gfCNCPoint5[20423] = {X 281.5052, Y 41.6984, Z -7.1667, A 0.000, B 0.000, C 0.000 }
gfCNCPoint5[20424] = {X 282.1444, Y 41.0612, Z -7.1667, A 0.000, B 0.000, C 0.000 }
gfCNCPoint5[20425] = {X 282.1444, Y 28.5919, Z -7.1667, A 0.000, B 0.000, C 0.000 }
gfCNCPoint5[20426] = {X 278.0644, Y 28.5919, Z -7.1667, A 0.000, B 0.000, C 0.000 }
gfCNCPoint5[20427] = {X 278.0644, Y 28.5919, Z -4.1667, A 0.000, B 0.000, C 0.000 }
gfCNCPoint5[20428] = {X 278.0644, Y 28.5919, Z 11.0000, A 0.000, B 0.000, C 0.000 }
gfCNCPoint5[20429] = {X 353.3540, Y 107.0415, Z 11.0000, A 0.000, B 0.000, C 0.000 }
gfCNCPoint5[20430] = {X 353.3540, Y 107.0415, Z -4.1667, A 0.000, B 0.000, C 0.000 }
gfCNCPoint5[20431] = {X 353.3540, Y 107.0415, Z -7.1667, A 0.000, B 0.000, C 0.000 }
gfCNCPoint5[20432] = {X 353.2425, Y 102.9631, Z -7.1667, A 0.000, B 0.000, C 0.000 }
gfCNCPoint5[20433] = {X 348.1839, Y 103.0329, Z -7.1667, A 0.000, B 0.000, C 0.000 }
gfCNCPoint5[20434] = {X 343.1251, Y 102.9662, Z -7.1667, A 0.000, B 0.000, C 0.000 }
gfCNCPoint5[20435] = {X 338.0701, Y 102.7628, Z -7.1667, A 0.000, B 0.000, C 0.000 }
gfCNCPoint5[20436] = {X 334.1158, Y 102.4859, Z -7.1667, A 0.000, B 0.000, C 0.000 }
gfCNCPoint5[20437] = {X 330.1765, Y 102.0440, Z -7.1667, A 0.000, B 0.000, C 0.000 }
gfCNCPoint5[20438] = {X 326.2592, Y 101.4380, Z -7.1667, A 0.000, B 0.000, C 0.000 }
gfCNCPoint5[20439] = {X 323.4097, Y 100.8332, Z -7.1667, A 0.000, B 0.000, C 0.000 }
gfCNCPoint5[20440] = {X 320.6125, Y 100.0203, Z -7.1667, A 0.000, B 0.000, C 0.000 }
gfCNCPoint5[20441] = {X 317.8826, Y 99.0038, Z -7.1667, A 0.000, B 0.000, C 0.000 }
gfCNCPoint5[20442] = {X 316.3697, Y 98.3059, Z -7.1667, A 0.000, B 0.000, C 0.000 }
gfCNCPoint5[20443] = {X 314.9204, Y 97.4840, Z -7.1667, A 0.000, B 0.000, C 0.000 }
gfCNCPoint5[20444] = {X 313.5448, Y 96.5439, Z -7.1667, A 0.000, B 0.000, C 0.000 }
gfCNCPoint5[20445] = {X 312.2527, Y 95.4921, Z -7.1667, A 0.000, B 0.000, C 0.000 }
gfCNCPoint5[20446] = {X 311.2489, Y 94.4933, Z -7.1667, A 0.000, B 0.000, C 0.000 }
gfCNCPoint5[20447] = {X 310.3705, Y 93.3827, Z -7.1667, A 0.000, B 0.000, C 0.000 }
gfCNCPoint5[20448] = {X 309.6299, Y 92.1758, Z -7.1667, A 0.000, B 0.000, C 0.000 }
gfCNCPoint5[20449] = {X 309.0375, Y 90.8896, Z -7.1667, A 0.000, B 0.000, C 0.000 }
gfCNCPoint5[20450] = {X 308.6017, Y 89.5424, Z -7.1667, A 0.000, B 0.000, C 0.000 }
gfCNCPoint5[20451] = {X 308.2582, Y 87.9192, Z -7.1667, A 0.000, B 0.000, C 0.000 }
gfCNCPoint5[20452] = {X 308.0553, Y 86.2726, Z -7.1667, A 0.000, B 0.000, C 0.000 }
gfCNCPoint5[20453] = {X 307.9944, Y 84.6146, Z -7.1667, A 0.000, B 0.000, C 0.000 }
gfCNCPoint5[20454] = {X 307.9956, Y 63.2121, Z -7.1667, A 0.000, B 0.000, C 0.000 }
gfCNCPoint5[20455] = {X 307.1443, Y 63.0028, Z -7.1667, A 0.000, B 0.000, C 0.000 }
gfCNCPoint5[20456] = {X 306.3527, Y 62.6258, Z -7.1667, A 0.000, B 0.000, C 0.000 }
gfCNCPoint5[20457] = {X 305.6536, Y 62.0968, Z -7.1667, A 0.000, B 0.000, C 0.000 }
gfCNCPoint5[20458] = {X 305.0756, Y 61.4376, Z -7.1667, A 0.000, B 0.000, C 0.000 }
gfCNCPoint5[20459] = {X 304.6427, Y 60.6752, Z -7.1667, A 0.000, B 0.000, C 0.000 }
gfCNCPoint5[20460] = {X 304.3725, Y 59.8412, Z -7.1667, A 0.000, B 0.000, C 0.000 }
gfCNCPoint5[20461] = {X 304.2764, Y 58.9697, Z -7.1667, A 0.000, B 0.000, C 0.000 }
gfCNCPoint5[20462] = {X 304.2762, Y 58.0000, Z -7.1667, A 0.000, B 0.000, C 0.000 }
gfCNCPoint5[20463] = {X 304.3845, Y 57.0387, Z -7.1667, A 0.000, B 0.000, C 0.000 }
gfCNCPoint5[20464] = {X 304.7040, Y 56.1256, Z -7.1667, A 0.000, B 0.000, C 0.000 }
gfCNCPoint5[20465] = {X 305.2187, Y 55.3065, Z -7.1667, A 0.000, B 0.000, C 0.000 }
gfCNCPoint5[20466] = {X 305.9027, Y 54.6225, Z -7.1667, A 0.000, B 0.000, C 0.000 }
gfCNCPoint5[20467] = {X 306.7218, Y 54.1078, Z -7.1667, A 0.000, B 0.000, C 0.000 }
gfCNCPoint5[20468] = {X 307.6349, Y 53.7883, Z -7.1667, A 0.000, B 0.000, C 0.000 }
gfCNCPoint5[20469] = {X 308.5962, Y 53.6800, Z -7.1667, A 0.000, B 0.000, C 0.000 }
gfCNCPoint5[20470] = {X 324.3107, Y 53.6800, Z -7.1667, A 0.000, B 0.000, C 0.000 }
gfCNCPoint5[20471] = {X 325.2720, Y 53.7883, Z -7.1667, A 0.000, B 0.000, C 0.000 }
gfCNCPoint5[20472] = {X 326.1851, Y 54.1078, Z -7.1667, A 0.000, B 0.000, C 0.000 }
gfCNCPoint5[20473] = {X 327.0042, Y 54.6225, Z -7.1667, A 0.000, B 0.000, C 0.000 }
gfCNCPoint5[20474] = {X 327.6882, Y 55.3065, Z -7.1667, A 0.000, B 0.000, C 0.000 }
gfCNCPoint5[20475] = {X 328.2029, Y 56.1256, Z -7.1667, A 0.000, B 0.000, C 0.000 }
gfCNCPoint5[20476] = {X 328.5224, Y 57.0387, Z -7.1667, A 0.000, B 0.000, C 0.000 }
gfCNCPoint5[20477] = {X 328.6307, Y 58.0000, Z -7.1667, A 0.000, B 0.000, C 0.000 }
gfCNCPoint5[20478] = {X 328.6307, Y 58.9358, Z -7.1667, A 0.000, B 0.000, C 0.000 }
gfCNCPoint5[20479] = {X 328.5369, Y 59.8122, Z -7.1667, A 0.000, B 0.000, C 0.000 }
gfCNCPoint5[20480] = {X 328.2687, Y 60.6517, Z -7.1667, A 0.000, B 0.000, C 0.000 }
gfCNCPoint5[20481] = {X 327.8370, Y 61.4202, Z -7.1667, A 0.000, B 0.000, C 0.000 }
gfCNCPoint5[20482] = {X 327.2595, Y 62.0860, Z -7.1667, A 0.000, B 0.000, C 0.000 }
gfCNCPoint5[20483] = {X 326.5599, Y 62.6220, Z -7.1667, A 0.000, B 0.000, C 0.000 }
gfCNCPoint5[20484] = {X 325.7666, Y 63.0063, Z -7.1667, A 0.000, B 0.000, C 0.000 }
gfCNCPoint5[20485] = {X 324.9123, Y 63.2230, Z -7.1667, A 0.000, B 0.000, C 0.000 }
gfCNCPoint5[20486] = {X 324.9142, Y 83.2295, Z -7.1667, A 0.000, B 0.000, C 0.000 }
gfCNCPoint5[20487] = {X 324.9278, Y 84.6145, Z -7.1667, A 0.000, B 0.000, C 0.000 }
gfCNCPoint5[20488] = {X 325.0045, Y 85.8430, Z -7.1667, A 0.000, B 0.000, C 0.000 }
gfCNCPoint5[20489] = {X 325.2231, Y 87.0543, Z -7.1667, A 0.000, B 0.000, C 0.000 }
gfCNCPoint5[20490] = {X 325.6723, Y 87.4784, Z -7.1667, A 0.000, B 0.000, C 0.000 }
gfCNCPoint5[20491] = {X 326.2083, Y 87.7855, Z -7.1667, A 0.000, B 0.000, C 0.000 }
gfCNCPoint5[20492] = {X 327.9881, Y 88.4971, Z -7.1667, A 0.000, B 0.000, C 0.000 }
gfCNCPoint5[20493] = {X 329.8404, Y 88.9900, Z -7.1667, A 0.000, B 0.000, C 0.000 }
gfCNCPoint5[20494] = {X 332.9245, Y 89.5434, Z -7.1667, A 0.000, B 0.000, C 0.000 }
gfCNCPoint5[20495] = {X 336.0365, Y 89.9077, Z -7.1667, A 0.000, B 0.000, C 0.000 }
gfCNCPoint5[20496] = {X 340.4063, Y 90.2019, Z -7.1667, A 0.000, B 0.000, C 0.000 }
gfCNCPoint5[20497] = {X 344.7832, Y 90.3557, Z -7.1667, A 0.000, B 0.000, C 0.000 }
gfCNCPoint5[20498] = {X 349.1628, Y 90.3690, Z -7.1667, A 0.000, B 0.000, C 0.000 }
gfCNCPoint5[20499] = {X 353.3143, Y 90.3007, Z -7.1667, A 0.000, B 0.000, C 0.000 }
gfCNCPoint5[20500] = {X 357.4606, Y 90.0817, Z -7.1667, A 0.000, B 0.000, C 0.000 }
gfCNCPoint5[20501] = {X 361.5962, Y 89.7124, Z -7.1667, A 0.000, B 0.000, C 0.000 }
gfCNCPoint5[20502] = {X 363.6775, Y 89.4253, Z -7.1667, A 0.000, B 0.000, C 0.000 }
gfCNCPoint5[20503] = {X 365.7396, Y 89.0233, Z -7.1667, A 0.000, B 0.000, C 0.000 }
gfCNCPoint5[20504] = {X 367.7763, Y 88.5076, Z -7.1667, A 0.000, B 0.000, C 0.000 }
gfCNCPoint5[20505] = {X 368.7088, Y 88.1946, Z -7.1667, A 0.000, B 0.000, C 0.000 }
gfCNCPoint5[20506] = {X 369.6001, Y 87.7787, Z -7.1667, A 0.000, B 0.000, C 0.000 }
gfCNCPoint5[20507] = {X 370.4388, Y 87.2650, Z -7.1667, A 0.000, B 0.000, C 0.000 }
gfCNCPoint5[20508] = {X 370.5874, Y 87.1102, Z -7.1667, A 0.000, B 0.000, C 0.000 }
gfCNCPoint5[20509] = {X 370.6640, Y 86.9098, Z -7.1667, A 0.000, B 0.000, C 0.000 }
gfCNCPoint5[20510] = {X 370.8553, Y 85.3746, Z -7.1667, A 0.000, B 0.000, C 0.000 }
gfCNCPoint5[20511] = {X 370.9191, Y 83.8288, Z -7.1667, A 0.000, B 0.000, C 0.000 }
gfCNCPoint5[20512] = {X 370.9200, Y 63.2123, Z -7.1667, A 0.000, B 0.000, C 0.000 }
gfCNCPoint5[20513] = {X 370.0684, Y 63.0031, Z -7.1667, A 0.000, B 0.000, C 0.000 }
gfCNCPoint5[20514] = {X 369.2766, Y 62.6263, Z -7.1667, A 0.000, B 0.000, C 0.000 }
gfCNCPoint5[20515] = {X 368.5772, Y 62.0973, Z -7.1667, A 0.000, B 0.000, C 0.000 }
gfCNCPoint5[20516] = {X 367.9990, Y 61.4381, Z -7.1667, A 0.000, B 0.000, C 0.000 }
gfCNCPoint5[20517] = {X 367.5659, Y 60.6756, Z -7.1667, A 0.000, B 0.000, C 0.000 }
gfCNCPoint5[20518] = {X 367.2956, Y 59.8414, Z -7.1667, A 0.000, B 0.000, C 0.000 }
gfCNCPoint5[20519] = {X 367.1994, Y 58.9697, Z -7.1667, A 0.000, B 0.000, C 0.000 }
gfCNCPoint5[20520] = {X 367.1993, Y 58.0000, Z -7.1667, A 0.000, B 0.000, C 0.000 }
gfCNCPoint5[20521] = {X 367.3076, Y 57.0387, Z -7.1667, A 0.000, B 0.000, C 0.000 }
gfCNCPoint5[20522] = {X 367.6271, Y 56.1256, Z -7.1667, A 0.000, B 0.000, C 0.000 }
gfCNCPoint5[20523] = {X 368.1418, Y 55.3065, Z -7.1667, A 0.000, B 0.000, C 0.000 }
gfCNCPoint5[20524] = {X 368.8258, Y 54.6225, Z -7.1667, A 0.000, B 0.000, C 0.000 }
gfCNCPoint5[20525] = {X 369.6449, Y 54.1078, Z -7.1667, A 0.000, B 0.000, C 0.000 }
gfCNCPoint5[20526] = {X 370.5580, Y 53.7883, Z -7.1667, A 0.000, B 0.000, C 0.000 }
gfCNCPoint5[20527] = {X 371.5193, Y 53.6800, Z -7.1667, A 0.000, B 0.000, C 0.000 }
gfCNCPoint5[20528] = {X 388.0597, Y 53.6800, Z -7.1667, A 0.000, B 0.000, C 0.000 }
gfCNCPoint5[20529] = {X 389.0210, Y 53.7883, Z -7.1667, A 0.000, B 0.000, C 0.000 }
gfCNCPoint5[20530] = {X 389.9341, Y 54.1078, Z -7.1667, A 0.000, B 0.000, C 0.000 }
gfCNCPoint5[20531] = {X 390.7532, Y 54.6225, Z -7.1667, A 0.000, B 0.000, C 0.000 }
gfCNCPoint5[20532] = {X 391.4372, Y 55.3065, Z -7.1667, A 0.000, B 0.000, C 0.000 }
gfCNCPoint5[20533] = {X 391.9519, Y 56.1256, Z -7.1667, A 0.000, B 0.000, C 0.000 }
gfCNCPoint5[20534] = {X 392.2714, Y 57.0387, Z -7.1667, A 0.000, B 0.000, C 0.000 }
gfCNCPoint5[20535] = {X 392.3797, Y 58.0000, Z -7.1667, A 0.000, B 0.000, C 0.000 }
gfCNCPoint5[20536] = {X 392.3797, Y 58.9342, Z -7.1667, A 0.000, B 0.000, C 0.000 }
gfCNCPoint5[20537] = {X 392.2681, Y 59.9098, Z -7.1667, A 0.000, B 0.000, C 0.000 }
gfCNCPoint5[20538] = {X 391.9390, Y 60.8349, Z -7.1667, A 0.000, B 0.000, C 0.000 }
gfCNCPoint5[20539] = {X 391.4969, Y 61.5528, Z -7.1667, A 0.000, B 0.000, C 0.000 }
gfCNCPoint5[20540] = {X 390.9244, Y 62.1718, Z -7.1667, A 0.000, B 0.000, C 0.000 }
gfCNCPoint5[20541] = {X 390.2431, Y 62.6686, Z -7.1667, A 0.000, B 0.000, C 0.000 }
gfCNCPoint5[20542] = {X 389.4787, Y 63.0243, Z -7.1667, A 0.000, B 0.000, C 0.000 }
gfCNCPoint5[20543] = {X 388.6600, Y 63.2257, Z -7.1667, A 0.000, B 0.000, C 0.000 }
gfCNCPoint5[20544] = {X 388.6579, Y 84.6147, Z -7.1667, A 0.000, B 0.000, C 0.000 }
gfCNCPoint5[20545] = {X 388.5980, Y 86.2730, Z -7.1667, A 0.000, B 0.000, C 0.000 }
gfCNCPoint5[20546] = {X 388.3937, Y 87.9198, Z -7.1667, A 0.000, B 0.000, C 0.000 }
gfCNCPoint5[20547] = {X 388.0465, Y 89.5425, Z -7.1667, A 0.000, B 0.000, C 0.000 }
gfCNCPoint5[20548] = {X 387.5140, Y 91.1297, Z -7.1667, A 0.000, B 0.000, C 0.000 }
gfCNCPoint5[20549] = {X 386.7643, Y 92.6265, Z -7.1667, A 0.000, B 0.000, C 0.000 }
gfCNCPoint5[20550] = {X 385.8124, Y 94.0036, Z -7.1667, A 0.000, B 0.000, C 0.000 }
gfCNCPoint5[20551] = {X 384.6769, Y 95.2337, Z -7.1667, A 0.000, B 0.000, C 0.000 }
gfCNCPoint5[20552] = {X 383.1622, Y 96.5103, Z -7.1667, A 0.000, B 0.000, C 0.000 }
gfCNCPoint5[20553] = {X 381.5205, Y 97.6188, Z -7.1667, A 0.000, B 0.000, C 0.000 }
gfCNCPoint5[20554] = {X 379.7703, Y 98.5466, Z -7.1667, A 0.000, B 0.000, C 0.000 }
gfCNCPoint5[20555] = {X 377.4988, Y 99.5016, Z -7.1667, A 0.000, B 0.000, C 0.000 }
gfCNCPoint5[20556] = {X 375.1648, Y 100.2918, Z -7.1667, A 0.000, B 0.000, C 0.000 }
gfCNCPoint5[20557] = {X 372.7804, Y 100.9132, Z -7.1667, A 0.000, B 0.000, C 0.000 }
gfCNCPoint5[20558] = {X 368.8695, Y 101.6665, Z -7.1667, A 0.000, B 0.000, C 0.000 }
gfCNCPoint5[20559] = {X 364.9264, Y 102.2268, Z -7.1667, A 0.000, B 0.000, C 0.000 }
gfCNCPoint5[20560] = {X 360.9605, Y 102.5928, Z -7.1667, A 0.000, B 0.000, C 0.000 }
gfCNCPoint5[20561] = {X 357.1034, Y 102.8177, Z -7.1667, A 0.000, B 0.000, C 0.000 }
gfCNCPoint5[20562] = {X 353.2425, Y 102.9631, Z -7.1667, A 0.000, B 0.000, C 0.000 }
gfCNCPoint5[20563] = {X 353.3518, Y 106.9616, Z -7.1667, A 0.000, B 0.000, C 0.000 }
gfCNCPoint5[20564] = {X 353.2403, Y 102.8831, Z -7.1667, A 0.000, B 0.000, C 0.000 }
gfCNCPoint5[20565] = {X 348.1838, Y 102.9529, Z -7.1667, A 0.000, B 0.000, C 0.000 }
gfCNCPoint5[20566] = {X 343.1272, Y 102.8862, Z -7.1667, A 0.000, B 0.000, C 0.000 }
gfCNCPoint5[20567] = {X 338.0742, Y 102.6829, Z -7.1667, A 0.000, B 0.000, C 0.000 }
gfCNCPoint5[20568] = {X 334.1232, Y 102.4062, Z -7.1667, A 0.000, B 0.000, C 0.000 }
gfCNCPoint5[20569] = {X 330.1871, Y 101.9647, Z -7.1667, A 0.000, B 0.000, C 0.000 }
gfCNCPoint5[20570] = {X 326.2730, Y 101.3592, Z -7.1667, A 0.000, B 0.000, C 0.000 }
gfCNCPoint5[20571] = {X 323.4292, Y 100.7556, Z -7.1667, A 0.000, B 0.000, C 0.000 }
gfCNCPoint5[20572] = {X 320.6375, Y 99.9443, Z -7.1667, A 0.000, B 0.000, C 0.000 }
gfCNCPoint5[20573] = {X 317.9131, Y 98.9298, Z -7.1667, A 0.000, B 0.000, C 0.000 }
gfCNCPoint5[20574] = {X 316.4062, Y 98.2347, Z -7.1667, A 0.000, B 0.000, C 0.000 }
gfCNCPoint5[20575] = {X 314.9627, Y 97.4161, Z -7.1667, A 0.000, B 0.000, C 0.000 }
gfCNCPoint5[20576] = {X 313.5926, Y 96.4797, Z -7.1667, A 0.000, B 0.000, C 0.000 }
gfCNCPoint5[20577] = {X 312.3056, Y 95.4321, Z -7.1667, A 0.000, B 0.000, C 0.000 }
gfCNCPoint5[20578] = {X 311.3086, Y 94.4401, Z -7.1667, A 0.000, B 0.000, C 0.000 }
gfCNCPoint5[20579] = {X 310.4361, Y 93.3368, Z -7.1667, A 0.000, B 0.000, C 0.000 }
gfCNCPoint5[20580] = {X 309.7005, Y 92.1380, Z -7.1667, A 0.000, B 0.000, C 0.000 }
gfCNCPoint5[20581] = {X 309.1121, Y 90.8605, Z -7.1667, A 0.000, B 0.000, C 0.000 }
gfCNCPoint5[20582] = {X 308.6791, Y 89.5223, Z -7.1667, A 0.000, B 0.000, C 0.000 }
gfCNCPoint5[20583] = {X 308.3371, Y 87.9059, Z -7.1667, A 0.000, B 0.000, C 0.000 }
gfCNCPoint5[20584] = {X 308.1350, Y 86.2661, Z -7.1667, A 0.000, B 0.000, C 0.000 }
gfCNCPoint5[20585] = {X 308.0744, Y 84.6150, Z -7.1667, A 0.000, B 0.000, C 0.000 }
gfCNCPoint5[20586] = {X 308.0756, Y 63.1420, Z -7.1667, A 0.000, B 0.000, C 0.000 }
gfCNCPoint5[20587] = {X 307.2274, Y 62.9470, Z -7.1667, A 0.000, B 0.000, C 0.000 }
gfCNCPoint5[20588] = {X 306.4368, Y 62.5830, Z -7.1667, A 0.000, B 0.000, C 0.000 }
gfCNCPoint5[20589] = {X 305.7373, Y 62.0652, Z -7.1667, A 0.000, B 0.000, C 0.000 }
gfCNCPoint5[20590] = {X 305.1581, Y 61.4154, Z -7.1667, A 0.000, B 0.000, C 0.000 }
gfCNCPoint5[20591] = {X 304.7239, Y 60.6611, Z -7.1667, A 0.000, B 0.000, C 0.000 }
gfCNCPoint5[20592] = {X 304.4528, Y 59.8341, Z -7.1667, A 0.000, B 0.000, C 0.000 }
gfCNCPoint5[20593] = {X 304.3564, Y 58.9691, Z -7.1667, A 0.000, B 0.000, C 0.000 }
gfCNCPoint5[20594] = {X 304.3562, Y 58.0000, Z -7.1667, A 0.000, B 0.000, C 0.000 }
gfCNCPoint5[20595] = {X 304.4625, Y 57.0565, Z -7.1667, A 0.000, B 0.000, C 0.000 }
gfCNCPoint5[20596] = {X 304.7761, Y 56.1603, Z -7.1667, A 0.000, B 0.000, C 0.000 }
gfCNCPoint5[20597] = {X 305.2813, Y 55.3564, Z -7.1667, A 0.000, B 0.000, C 0.000 }
gfCNCPoint5[20598] = {X 305.9526, Y 54.6850, Z -7.1667, A 0.000, B 0.000, C 0.000 }
gfCNCPoint5[20599] = {X 306.7566, Y 54.1799, Z -7.1667, A 0.000, B 0.000, C 0.000 }
gfCNCPoint5[20600] = {X 307.6527, Y 53.8663, Z -7.1667, A 0.000, B 0.000, C 0.000 }
gfCNCPoint5[20601] = {X 308.5962, Y 53.7600, Z -7.1667, A 0.000, B 0.000, C 0.000 }
gfCNCPoint5[20602] = {X 324.3107, Y 53.7600, Z -7.1667, A 0.000, B 0.000, C 0.000 }
gfCNCPoint5[20603] = {X 325.2542, Y 53.8663, Z -7.1667, A 0.000, B 0.000, C 0.000 }
gfCNCPoint5[20604] = {X 326.1504, Y 54.1799, Z -7.1667, A 0.000, B 0.000, C 0.000 }
gfCNCPoint5[20605] = {X 326.9543, Y 54.6850, Z -7.1667, A 0.000, B 0.000, C 0.000 }
gfCNCPoint5[20606] = {X 327.6257, Y 55.3564, Z -7.1667, A 0.000, B 0.000, C 0.000 }
gfCNCPoint5[20607] = {X 328.1308, Y 56.1603, Z -7.1667, A 0.000, B 0.000, C 0.000 }
gfCNCPoint5[20608] = {X 328.4444, Y 57.0565, Z -7.1667, A 0.000, B 0.000, C 0.000 }
gfCNCPoint5[20609] = {X 328.5507, Y 58.0000, Z -7.1667, A 0.000, B 0.000, C 0.000 }
gfCNCPoint5[20610] = {X 328.5507, Y 58.9354, Z -7.1667, A 0.000, B 0.000, C 0.000 }
gfCNCPoint5[20611] = {X 328.4566, Y 59.8053, Z -7.1667, A 0.000, B 0.000, C 0.000 }
gfCNCPoint5[20612] = {X 328.1875, Y 60.6379, Z -7.1667, A 0.000, B 0.000, C 0.000 }
gfCNCPoint5[20613] = {X 327.7545, Y 61.3982, Z -7.1667, A 0.000, B 0.000, C 0.000 }
gfCNCPoint5[20614] = {X 327.1759, Y 62.0546, Z -7.1667, A 0.000, B 0.000, C 0.000 }
gfCNCPoint5[20615] = {X 326.4758, Y 62.5795, Z -7.1667, A 0.000, B 0.000, C 0.000 }
gfCNCPoint5[20616] = {X 325.6836, Y 62.9510, Z -7.1667, A 0.000, B 0.000, C 0.000 }
gfCNCPoint5[20617] = {X 324.8323, Y 63.1534, Z -7.1667, A 0.000, B 0.000, C 0.000 }
gfCNCPoint5[20618] = {X 324.8342, Y 83.2300, Z -7.1667, A 0.000, B 0.000, C 0.000 }
gfCNCPoint5[20619] = {X 324.8478, Y 84.6149, Z -7.1667, A 0.000, B 0.000, C 0.000 }
gfCNCPoint5[20620] = {X 324.9262, Y 85.8619, Z -7.1667, A 0.000, B 0.000, C 0.000 }
gfCNCPoint5[20621] = {X 325.1497, Y 87.0911, Z -7.1667, A 0.000, B 0.000, C 0.000 }
gfCNCPoint5[20622] = {X 325.6165, Y 87.5366, Z -7.1667, A 0.000, B 0.000, C 0.000 }
gfCNCPoint5[20623] = {X 326.1756, Y 87.8585, Z -7.1667, A 0.000, B 0.000, C 0.000 }
gfCNCPoint5[20624] = {X 327.9636, Y 88.5733, Z -7.1667, A 0.000, B 0.000, C 0.000 }
gfCNCPoint5[20625] = {X 329.8245, Y 89.0685, Z -7.1667, A 0.000, B 0.000, C 0.000 }
gfCNCPoint5[20626] = {X 332.9131, Y 89.6226, Z -7.1667, A 0.000, B 0.000, C 0.000 }
gfCNCPoint5[20627] = {X 336.0297, Y 89.9874, Z -7.1667, A 0.000, B 0.000, C 0.000 }
gfCNCPoint5[20628] = {X 340.4020, Y 90.2818, Z -7.1667, A 0.000, B 0.000, C 0.000 }
gfCNCPoint5[20629] = {X 344.7816, Y 90.4357, Z -7.1667, A 0.000, B 0.000, C 0.000 }
gfCNCPoint5[20630] = {X 349.1638, Y 90.4490, Z -7.1667, A 0.000, B 0.000, C 0.000 }
gfCNCPoint5[20631] = {X 353.3179, Y 90.3806, Z -7.1667, A 0.000, B 0.000, C 0.000 }
gfCNCPoint5[20632] = {X 357.4668, Y 90.1615, Z -7.1667, A 0.000, B 0.000, C 0.000 }
gfCNCPoint5[20633] = {X 361.6050, Y 89.7919, Z -7.1667, A 0.000, B 0.000, C 0.000 }
gfCNCPoint5[20634] = {X 363.6906, Y 89.5042, Z -7.1667, A 0.000, B 0.000, C 0.000 }
gfCNCPoint5[20635] = {X 365.7571, Y 89.1014, Z -7.1667, A 0.000, B 0.000, C 0.000 }
gfCNCPoint5[20636] = {X 367.7981, Y 88.5846, Z -7.1667, A 0.000, B 0.000, C 0.000 }
gfCNCPoint5[20637] = {X 368.7389, Y 88.2688, Z -7.1667, A 0.000, B 0.000, C 0.000 }
gfCNCPoint5[20638] = {X 369.6381, Y 87.8490, Z -7.1667, A 0.000, B 0.000, C 0.000 }
gfCNCPoint5[20639] = {X 370.4844, Y 87.3307, Z -7.1667, A 0.000, B 0.000, C 0.000 }
gfCNCPoint5[20640] = {X 370.6550, Y 87.1530, Z -7.1667, A 0.000, B 0.000, C 0.000 }
gfCNCPoint5[20641] = {X 370.7429, Y 86.9229, Z -7.1667, A 0.000, B 0.000, C 0.000 }
gfCNCPoint5[20642] = {X 370.9350, Y 85.3812, Z -7.1667, A 0.000, B 0.000, C 0.000 }
gfCNCPoint5[20643] = {X 370.9991, Y 83.8288, Z -7.1667, A 0.000, B 0.000, C 0.000 }
gfCNCPoint5[20644] = {X 371.0000, Y 63.1421, Z -7.1667, A 0.000, B 0.000, C 0.000 }
gfCNCPoint5[20645] = {X 370.1515, Y 62.9474, Z -7.1667, A 0.000, B 0.000, C 0.000 }
gfCNCPoint5[20646] = {X 369.3607, Y 62.5835, Z -7.1667, A 0.000, B 0.000, C 0.000 }
gfCNCPoint5[20647] = {X 368.6609, Y 62.0657, Z -7.1667, A 0.000, B 0.000, C 0.000 }
gfCNCPoint5[20648] = {X 368.0815, Y 61.4159, Z -7.1667, A 0.000, B 0.000, C 0.000 }
gfCNCPoint5[20649] = {X 367.6471, Y 60.6615, Z -7.1667, A 0.000, B 0.000, C 0.000 }
gfCNCPoint5[20650] = {X 367.3759, Y 59.8343, Z -7.1667, A 0.000, B 0.000, C 0.000 }
gfCNCPoint5[20651] = {X 367.2794, Y 58.9691, Z -7.1667, A 0.000, B 0.000, C 0.000 }
gfCNCPoint5[20652] = {X 367.2793, Y 58.0000, Z -7.1667, A 0.000, B 0.000, C 0.000 }
gfCNCPoint5[20653] = {X 367.3856, Y 57.0565, Z -7.1667, A 0.000, B 0.000, C 0.000 }
gfCNCPoint5[20654] = {X 367.6992, Y 56.1603, Z -7.1667, A 0.000, B 0.000, C 0.000 }
gfCNCPoint5[20655] = {X 368.2043, Y 55.3564, Z -7.1667, A 0.000, B 0.000, C 0.000 }
gfCNCPoint5[20656] = {X 368.8757, Y 54.6850, Z -7.1667, A 0.000, B 0.000, C 0.000 }
gfCNCPoint5[20657] = {X 369.6796, Y 54.1799, Z -7.1667, A 0.000, B 0.000, C 0.000 }
gfCNCPoint5[20658] = {X 370.5758, Y 53.8663, Z -7.1667, A 0.000, B 0.000, C 0.000 }
gfCNCPoint5[20659] = {X 371.5193, Y 53.7600, Z -7.1667, A 0.000, B 0.000, C 0.000 }
gfCNCPoint5[20660] = {X 388.0597, Y 53.7600, Z -7.1667, A 0.000, B 0.000, C 0.000 }
gfCNCPoint5[20661] = {X 389.0032, Y 53.8663, Z -7.1667, A 0.000, B 0.000, C 0.000 }
gfCNCPoint5[20662] = {X 389.8993, Y 54.1799, Z -7.1667, A 0.000, B 0.000, C 0.000 }
gfCNCPoint5[20663] = {X 390.7033, Y 54.6850, Z -7.1667, A 0.000, B 0.000, C 0.000 }
gfCNCPoint5[20664] = {X 391.3746, Y 55.3564, Z -7.1667, A 0.000, B 0.000, C 0.000 }
gfCNCPoint5[20665] = {X 391.8798, Y 56.1603, Z -7.1667, A 0.000, B 0.000, C 0.000 }
gfCNCPoint5[20666] = {X 392.1934, Y 57.0565, Z -7.1667, A 0.000, B 0.000, C 0.000 }
gfCNCPoint5[20667] = {X 392.2997, Y 58.0000, Z -7.1667, A 0.000, B 0.000, C 0.000 }
gfCNCPoint5[20668] = {X 392.2997, Y 58.9342, Z -7.1667, A 0.000, B 0.000, C 0.000 }
gfCNCPoint5[20669] = {X 392.1901, Y 59.8917, Z -7.1667, A 0.000, B 0.000, C 0.000 }
gfCNCPoint5[20670] = {X 391.8672, Y 60.7997, Z -7.1667, A 0.000, B 0.000, C 0.000 }
gfCNCPoint5[20671] = {X 391.4248, Y 61.5154, Z -7.1667, A 0.000, B 0.000, C 0.000 }
gfCNCPoint5[20672] = {X 390.8506, Y 62.1304, Z -7.1667, A 0.000, B 0.000, C 0.000 }
gfCNCPoint5[20673] = {X 390.1667, Y 62.6205, Z -7.1667, A 0.000, B 0.000, C 0.000 }
gfCNCPoint5[20674] = {X 389.3999, Y 62.9669, Z -7.1667, A 0.000, B 0.000, C 0.000 }
gfCNCPoint5[20675] = {X 388.5800, Y 63.1559, Z -7.1667, A 0.000, B 0.000, C 0.000 }
gfCNCPoint5[20676] = {X 388.5779, Y 84.6150, Z -7.1667, A 0.000, B 0.000, C 0.000 }
gfCNCPoint5[20677] = {X 388.5183, Y 86.2665, Z -7.1667, A 0.000, B 0.000, C 0.000 }
gfCNCPoint5[20678] = {X 388.3148, Y 87.9064, Z -7.1667, A 0.000, B 0.000, C 0.000 }
gfCNCPoint5[20679] = {X 387.9691, Y 89.5224, Z -7.1667, A 0.000, B 0.000, C 0.000 }
gfCNCPoint5[20680] = {X 387.4401, Y 91.0989, Z -7.1667, A 0.000, B 0.000, C 0.000 }
gfCNCPoint5[20681] = {X 386.6955, Y 92.5857, Z -7.1667, A 0.000, B 0.000, C 0.000 }
gfCNCPoint5[20682] = {X 385.7500, Y 93.9536, Z -7.1667, A 0.000, B 0.000, C 0.000 }
gfCNCPoint5[20683] = {X 384.6221, Y 95.1754, Z -7.1667, A 0.000, B 0.000, C 0.000 }
gfCNCPoint5[20684] = {X 383.1139, Y 96.4465, Z -7.1667, A 0.000, B 0.000, C 0.000 }
gfCNCPoint5[20685] = {X 381.4793, Y 97.5502, Z -7.1667, A 0.000, B 0.000, C 0.000 }
gfCNCPoint5[20686] = {X 379.7366, Y 98.4740, Z -7.1667, A 0.000, B 0.000, C 0.000 }
gfCNCPoint5[20687] = {X 377.4704, Y 99.4268, Z -7.1667, A 0.000, B 0.000, C 0.000 }
gfCNCPoint5[20688] = {X 375.1419, Y 100.2151, Z -7.1667, A 0.000, B 0.000, C 0.000 }
gfCNCPoint5[20689] = {X 372.7630, Y 100.8351, Z -7.1667, A 0.000, B 0.000, C 0.000 }
gfCNCPoint5[20690] = {X 368.8561, Y 101.5876, Z -7.1667, A 0.000, B 0.000, C 0.000 }
gfCNCPoint5[20691] = {X 364.9169, Y 102.1473, Z -7.1667, A 0.000, B 0.000, C 0.000 }
gfCNCPoint5[20692] = {X 360.9550, Y 102.5130, Z -7.1667, A 0.000, B 0.000, C 0.000 }
gfCNCPoint5[20693] = {X 357.0996, Y 102.7378, Z -7.1667, A 0.000, B 0.000, C 0.000 }
gfCNCPoint5[20694] = {X 353.2403, Y 102.8831, Z -7.1667, A 0.000, B 0.000, C 0.000 }
gfCNCPoint5[20695] = {X 353.3496, Y 106.8816, Z -7.1667, A 0.000, B 0.000, C 0.000 }
gfCNCPoint5[20696] = {X 353.2382, Y 102.8031, Z -7.1667, A 0.000, B 0.000, C 0.000 }
gfCNCPoint5[20697] = {X 348.1837, Y 102.8729, Z -7.1667, A 0.000, B 0.000, C 0.000 }
gfCNCPoint5[20698] = {X 343.1292, Y 102.8062, Z -7.1667, A 0.000, B 0.000, C 0.000 }
gfCNCPoint5[20699] = {X 338.0783, Y 102.6030, Z -7.1667, A 0.000, B 0.000, C 0.000 }
gfCNCPoint5[20700] = {X 334.1305, Y 102.3266, Z -7.1667, A 0.000, B 0.000, C 0.000 }
gfCNCPoint5[20701] = {X 330.1977, Y 101.8854, Z -7.1667, A 0.000, B 0.000, C 0.000 }
gfCNCPoint5[20702] = {X 326.2868, Y 101.2804, Z -7.1667, A 0.000, B 0.000, C 0.000 }
gfCNCPoint5[20703] = {X 323.4487, Y 100.6780, Z -7.1667, A 0.000, B 0.000, C 0.000 }
gfCNCPoint5[20704] = {X 320.6626, Y 99.8683, Z -7.1667, A 0.000, B 0.000, C 0.000 }
gfCNCPoint5[20705] = {X 317.9436, Y 98.8558, Z -7.1667, A 0.000, B 0.000, C 0.000 }
gfCNCPoint5[20706] = {X 316.4427, Y 98.1635, Z -7.1667, A 0.000, B 0.000, C 0.000 }
gfCNCPoint5[20707] = {X 315.0050, Y 97.3482, Z -7.1667, A 0.000, B 0.000, C 0.000 }
gfCNCPoint5[20708] = {X 313.6404, Y 96.4156, Z -7.1667, A 0.000, B 0.000, C 0.000 }
gfCNCPoint5[20709] = {X 312.3586, Y 95.3722, Z -7.1667, A 0.000, B 0.000, C 0.000 }
gfCNCPoint5[20710] = {X 311.3683, Y 94.3868, Z -7.1667, A 0.000, B 0.000, C 0.000 }
gfCNCPoint5[20711] = {X 310.5017, Y 93.2910, Z -7.1667, A 0.000, B 0.000, C 0.000 }
gfCNCPoint5[20712] = {X 309.7710, Y 92.1003, Z -7.1667, A 0.000, B 0.000, C 0.000 }
gfCNCPoint5[20713] = {X 309.1866, Y 90.8314, Z -7.1667, A 0.000, B 0.000, C 0.000 }
gfCNCPoint5[20714] = {X 308.7565, Y 89.5023, Z -7.1667, A 0.000, B 0.000, C 0.000 }
gfCNCPoint5[20715] = {X 308.4159, Y 87.8925, Z -7.1667, A 0.000, B 0.000, C 0.000 }
gfCNCPoint5[20716] = {X 308.2147, Y 86.2595, Z -7.1667, A 0.000, B 0.000, C 0.000 }
gfCNCPoint5[20717] = {X 308.1544, Y 84.6152, Z -7.1667, A 0.000, B 0.000, C 0.000 }
gfCNCPoint5[20718] = {X 308.1556, Y 63.0707, Z -7.1667, A 0.000, B 0.000, C 0.000 }
gfCNCPoint5[20719] = {X 307.3107, Y 62.8904, Z -7.1667, A 0.000, B 0.000, C 0.000 }
gfCNCPoint5[20720] = {X 306.5212, Y 62.5396, Z -7.1667, A 0.000, B 0.000, C 0.000 }
gfCNCPoint5[20721] = {X 305.8211, Y 62.0332, Z -7.1667, A 0.000, B 0.000, C 0.000 }
gfCNCPoint5[20722] = {X 305.2408, Y 61.3931, Z -7.1667, A 0.000, B 0.000, C 0.000 }
gfCNCPoint5[20723] = {X 304.8052, Y 60.6470, Z -7.1667, A 0.000, B 0.000, C 0.000 }
gfCNCPoint5[20724] = {X 304.5332, Y 59.8270, Z -7.1667, A 0.000, B 0.000, C 0.000 }
gfCNCPoint5[20725] = {X 304.4364, Y 58.9684, Z -7.1667, A 0.000, B 0.000, C 0.000 }
gfCNCPoint5[20726] = {X 304.4362, Y 58.0000, Z -7.1667, A 0.000, B 0.000, C 0.000 }
gfCNCPoint5[20727] = {X 304.5405, Y 57.0743, Z -7.1667, A 0.000, B 0.000, C 0.000 }
gfCNCPoint5[20728] = {X 304.8482, Y 56.1950, Z -7.1667, A 0.000, B 0.000, C 0.000 }
gfCNCPoint5[20729] = {X 305.3438, Y 55.4063, Z -7.1667, A 0.000, B 0.000, C 0.000 }
gfCNCPoint5[20730] = {X 306.0025, Y 54.7476, Z -7.1667, A 0.000, B 0.000, C 0.000 }
gfCNCPoint5[20731] = {X 306.7913, Y 54.2520, Z -7.1667, A 0.000, B 0.000, C 0.000 }
gfCNCPoint5[20732] = {X 307.6705, Y 53.9443, Z -7.1667, A 0.000, B 0.000, C 0.000 }
gfCNCPoint5[20733] = {X 308.5962, Y 53.8400, Z -7.1667, A 0.000, B 0.000, C 0.000 }
gfCNCPoint5[20734] = {X 324.3107, Y 53.8400, Z -7.1667, A 0.000, B 0.000, C 0.000 }
gfCNCPoint5[20735] = {X 325.2364, Y 53.9443, Z -7.1667, A 0.000, B 0.000, C 0.000 }
gfCNCPoint5[20736] = {X 326.1156, Y 54.2520, Z -7.1667, A 0.000, B 0.000, C 0.000 }
gfCNCPoint5[20737] = {X 326.9044, Y 54.7476, Z -7.1667, A 0.000, B 0.000, C 0.000 }
gfCNCPoint5[20738] = {X 327.5631, Y 55.4063, Z -7.1667, A 0.000, B 0.000, C 0.000 }
gfCNCPoint5[20739] = {X 328.0587, Y 56.1950, Z -7.1667, A 0.000, B 0.000, C 0.000 }
gfCNCPoint5[20740] = {X 328.3664, Y 57.0743, Z -7.1667, A 0.000, B 0.000, C 0.000 }
gfCNCPoint5[20741] = {X 328.4707, Y 58.0000, Z -7.1667, A 0.000, B 0.000, C 0.000 }
gfCNCPoint5[20742] = {X 328.4707, Y 58.9349, Z -7.1667, A 0.000, B 0.000, C 0.000 }
gfCNCPoint5[20743] = {X 328.3763, Y 59.7984, Z -7.1667, A 0.000, B 0.000, C 0.000 }
gfCNCPoint5[20744] = {X 328.1061, Y 60.6239, Z -7.1667, A 0.000, B 0.000, C 0.000 }
gfCNCPoint5[20745] = {X 327.6719, Y 61.3761, Z -7.1667, A 0.000, B 0.000, C 0.000 }
gfCNCPoint5[20746] = {X 327.0921, Y 62.0229, Z -7.1667, A 0.000, B 0.000, C 0.000 }
gfCNCPoint5[20747] = {X 326.3916, Y 62.5365, Z -7.1667, A 0.000, B 0.000, C 0.000 }
gfCNCPoint5[20748] = {X 325.6004, Y 62.8948, Z -7.1667, A 0.000, B 0.000, C 0.000 }
gfCNCPoint5[20749] = {X 324.7523, Y 63.0827, Z -7.1667, A 0.000, B 0.000, C 0.000 }
gfCNCPoint5[20750] = {X 324.7542, Y 83.2304, Z -7.1667, A 0.000, B 0.000, C 0.000 }
gfCNCPoint5[20751] = {X 324.7678, Y 84.6152, Z -7.1667, A 0.000, B 0.000, C 0.000 }
gfCNCPoint5[20752] = {X 324.8479, Y 85.8806, Z -7.1667, A 0.000, B 0.000, C 0.000 }
gfCNCPoint5[20753] = {X 325.0763, Y 87.1277, Z -7.1667, A 0.000, B 0.000, C 0.000 }
gfCNCPoint5[20754] = {X 325.5606, Y 87.5946, Z -7.1667, A 0.000, B 0.000, C 0.000 }
gfCNCPoint5[20755] = {X 326.1428, Y 87.9315, Z -7.1667, A 0.000, B 0.000, C 0.000 }
gfCNCPoint5[20756] = {X 327.9392, Y 88.6494, Z -7.1667, A 0.000, B 0.000, C 0.000 }
gfCNCPoint5[20757] = {X 329.8086, Y 89.1469, Z -7.1667, A 0.000, B 0.000, C 0.000 }
gfCNCPoint5[20758] = {X 332.9017, Y 89.7017, Z -7.1667, A 0.000, B 0.000, C 0.000 }
gfCNCPoint5[20759] = {X 336.0229, Y 90.0671, Z -7.1667, A 0.000, B 0.000, C 0.000 }
gfCNCPoint5[20760] = {X 340.3978, Y 90.3617, Z -7.1667, A 0.000, B 0.000, C 0.000 }
gfCNCPoint5[20761] = {X 344.7800, Y 90.5157, Z -7.1667, A 0.000, B 0.000, C 0.000 }
gfCNCPoint5[20762] = {X 349.1649, Y 90.5290, Z -7.1667, A 0.000, B 0.000, C 0.000 }
gfCNCPoint5[20763] = {X 353.3215, Y 90.4605, Z -7.1667, A 0.000, B 0.000, C 0.000 }
gfCNCPoint5[20764] = {X 357.4730, Y 90.2412, Z -7.1667, A 0.000, B 0.000, C 0.000 }
gfCNCPoint5[20765] = {X 361.6137, Y 89.8714, Z -7.1667, A 0.000, B 0.000, C 0.000 }
gfCNCPoint5[20766] = {X 363.7037, Y 89.5831, Z -7.1667, A 0.000, B 0.000, C 0.000 }
gfCNCPoint5[20767] = {X 365.7746, Y 89.1794, Z -7.1667, A 0.000, B 0.000, C 0.000 }
gfCNCPoint5[20768] = {X 367.8199, Y 88.6616, Z -7.1667, A 0.000, B 0.000, C 0.000 }
gfCNCPoint5[20769] = {X 368.7690, Y 88.3429, Z -7.1667, A 0.000, B 0.000, C 0.000 }
gfCNCPoint5[20770] = {X 369.6762, Y 87.9194, Z -7.1667, A 0.000, B 0.000, C 0.000 }
gfCNCPoint5[20771] = {X 370.5300, Y 87.3965, Z -7.1667, A 0.000, B 0.000, C 0.000 }
gfCNCPoint5[20772] = {X 370.7225, Y 87.1958, Z -7.1667, A 0.000, B 0.000, C 0.000 }
gfCNCPoint5[20773] = {X 370.8218, Y 86.9361, Z -7.1667, A 0.000, B 0.000, C 0.000 }
gfCNCPoint5[20774] = {X 371.0147, Y 85.3878, Z -7.1667, A 0.000, B 0.000, C 0.000 }
gfCNCPoint5[20775] = {X 371.0791, Y 83.8288, Z -7.1667, A 0.000, B 0.000, C 0.000 }
gfCNCPoint5[20776] = {X 371.0800, Y 63.0708, Z -7.1667, A 0.000, B 0.000, C 0.000 }
gfCNCPoint5[20777] = {X 370.9773, Y 63.0586, Z -7.1667, A 0.000, B 0.000, C 0.000 }
gfCNCPoint5[20778] = {X 370.8750, Y 63.0439, Z -7.1667, A 0.000, B 0.000, C 0.000 }
gfCNCPoint5[20779] = {X 369.9377, Y 62.7817, Z -7.1667, A 0.000, B 0.000, C 0.000 }
gfCNCPoint5[20780] = {X 369.0869, Y 62.3089, Z -7.1667, A 0.000, B 0.000, C 0.000 }
gfCNCPoint5[20781] = {X 368.3693, Y 61.6513, Z -7.1667, A 0.000, B 0.000, C 0.000 }
gfCNCPoint5[20782] = {X 367.8242, Y 60.8450, Z -7.1667, A 0.000, B 0.000, C 0.000 }
gfCNCPoint5[20783] = {X 367.4813, Y 59.9341, Z -7.1667, A 0.000, B 0.000, C 0.000 }
gfCNCPoint5[20784] = {X 367.3594, Y 58.9684, Z -7.1667, A 0.000, B 0.000, C 0.000 }
gfCNCPoint5[20785] = {X 367.3593, Y 58.0000, Z -7.1667, A 0.000, B 0.000, C 0.000 }
gfCNCPoint5[20786] = {X 367.4636, Y 57.0743, Z -7.1667, A 0.000, B 0.000, C 0.000 }
gfCNCPoint5[20787] = {X 367.7713, Y 56.1950, Z -7.1667, A 0.000, B 0.000, C 0.000 }
gfCNCPoint5[20788] = {X 368.2669, Y 55.4063, Z -7.1667, A 0.000, B 0.000, C 0.000 }
gfCNCPoint5[20789] = {X 368.9256, Y 54.7476, Z -7.1667, A 0.000, B 0.000, C 0.000 }
gfCNCPoint5[20790] = {X 369.7143, Y 54.2520, Z -7.1667, A 0.000, B 0.000, C 0.000 }
gfCNCPoint5[20791] = {X 370.5936, Y 53.9443, Z -7.1667, A 0.000, B 0.000, C 0.000 }
gfCNCPoint5[20792] = {X 371.5193, Y 53.8400, Z -7.1667, A 0.000, B 0.000, C 0.000 }
gfCNCPoint5[20793] = {X 388.0597, Y 53.8400, Z -7.1667, A 0.000, B 0.000, C 0.000 }
gfCNCPoint5[20794] = {X 388.9854, Y 53.9443, Z -7.1667, A 0.000, B 0.000, C 0.000 }
gfCNCPoint5[20795] = {X 389.8646, Y 54.2520, Z -7.1667, A 0.000, B 0.000, C 0.000 }
gfCNCPoint5[20796] = {X 390.6534, Y 54.7476, Z -7.1667, A 0.000, B 0.000, C 0.000 }
gfCNCPoint5[20797] = {X 391.3121, Y 55.4063, Z -7.1667, A 0.000, B 0.000, C 0.000 }
gfCNCPoint5[20798] = {X 391.8077, Y 56.1950, Z -7.1667, A 0.000, B 0.000, C 0.000 }
gfCNCPoint5[20799] = {X 392.1154, Y 57.0743, Z -7.1667, A 0.000, B 0.000, C 0.000 }
gfCNCPoint5[20800] = {X 392.2197, Y 58.0000, Z -7.1667, A 0.000, B 0.000, C 0.000 }
gfCNCPoint5[20801] = {X 392.2197, Y 58.9342, Z -7.1667, A 0.000, B 0.000, C 0.000 }
gfCNCPoint5[20802] = {X 392.1122, Y 59.8736, Z -7.1667, A 0.000, B 0.000, C 0.000 }
gfCNCPoint5[20803] = {X 391.7953, Y 60.7645, Z -7.1667, A 0.000, B 0.000, C 0.000 }
gfCNCPoint5[20804] = {X 391.2528, Y 61.6015, Z -7.1667, A 0.000, B 0.000, C 0.000 }
gfCNCPoint5[20805] = {X 390.5276, Y 62.2862, Z -7.1667, A 0.000, B 0.000, C 0.000 }
gfCNCPoint5[20806] = {X 389.6609, Y 62.7799, Z -7.1667, A 0.000, B 0.000, C 0.000 }
gfCNCPoint5[20807] = {X 388.7019, Y 63.0543, Z -7.1667, A 0.000, B 0.000, C 0.000 }
gfCNCPoint5[20808] = {X 388.6017, Y 63.0692, Z -7.1667, A 0.000, B 0.000, C 0.000 }
gfCNCPoint5[20809] = {X 388.5011, Y 63.0816, Z -7.1667, A 0.000, B 0.000, C 0.000 }
gfCNCPoint5[20810] = {X 388.4979, Y 84.6154, Z -7.1667, A 0.000, B 0.000, C 0.000 }
gfCNCPoint5[20811] = {X 388.4386, Y 86.2600, Z -7.1667, A 0.000, B 0.000, C 0.000 }
gfCNCPoint5[20812] = {X 388.2359, Y 87.8931, Z -7.1667, A 0.000, B 0.000, C 0.000 }
gfCNCPoint5[20813] = {X 387.8916, Y 89.5023, Z -7.1667, A 0.000, B 0.000, C 0.000 }
gfCNCPoint5[20814] = {X 387.3663, Y 91.0682, Z -7.1667, A 0.000, B 0.000, C 0.000 }
gfCNCPoint5[20815] = {X 386.6267, Y 92.5450, Z -7.1667, A 0.000, B 0.000, C 0.000 }
gfCNCPoint5[20816] = {X 385.6875, Y 93.9036, Z -7.1667, A 0.000, B 0.000, C 0.000 }
gfCNCPoint5[20817] = {X 384.5673, Y 95.1172, Z -7.1667, A 0.000, B 0.000, C 0.000 }
gfCNCPoint5[20818] = {X 383.0656, Y 96.3827, Z -7.1667, A 0.000, B 0.000, C 0.000 }
gfCNCPoint5[20819] = {X 381.4381, Y 97.4816, Z -7.1667, A 0.000, B 0.000, C 0.000 }
gfCNCPoint5[20820] = {X 379.7030, Y 98.4014, Z -7.1667, A 0.000, B 0.000, C 0.000 }
gfCNCPoint5[20821] = {X 377.4420, Y 99.3520, Z -7.1667, A 0.000, B 0.000, C 0.000 }
gfCNCPoint5[20822] = {X 375.1189, Y 100.1385, Z -7.1667, A 0.000, B 0.000, C 0.000 }
gfCNCPoint5[20823] = {X 372.7456, Y 100.7571, Z -7.1667, A 0.000, B 0.000, C 0.000 }
gfCNCPoint5[20824] = {X 368.8426, Y 101.5088, Z -7.1667, A 0.000, B 0.000, C 0.000 }
gfCNCPoint5[20825] = {X 364.9074, Y 102.0679, Z -7.1667, A 0.000, B 0.000, C 0.000 }
gfCNCPoint5[20826] = {X 360.9496, Y 102.4332, Z -7.1667, A 0.000, B 0.000, C 0.000 }
gfCNCPoint5[20827] = {X 357.0958, Y 102.6579, Z -7.1667, A 0.000, B 0.000, C 0.000 }
gfCNCPoint5[20828] = {X 353.2382, Y 102.8031, Z -7.1667, A 0.000, B 0.000, C 0.000 }
gfCNCPoint5[20829] = {X 353.3474, Y 106.8016, Z -7.1667, A 0.000, B 0.000, C 0.000 }
gfCNCPoint5[20830] = {X 353.2360, Y 102.7232, Z -7.1667, A 0.000, B 0.000, C 0.000 }
gfCNCPoint5[20831] = {X 348.1836, Y 102.7929, Z -7.1667, A 0.000, B 0.000, C 0.000 }
gfCNCPoint5[20832] = {X 343.1312, Y 102.7262, Z -7.1667, A 0.000, B 0.000, C 0.000 }
gfCNCPoint5[20833] = {X 338.0825, Y 102.5231, Z -7.1667, A 0.000, B 0.000, C 0.000 }
gfCNCPoint5[20834] = {X 334.1379, Y 102.2469, Z -7.1667, A 0.000, B 0.000, C 0.000 }
gfCNCPoint5[20835] = {X 330.2084, Y 101.8061, Z -7.1667, A 0.000, B 0.000, C 0.000 }
gfCNCPoint5[20836] = {X 326.3007, Y 101.2016, Z -7.1667, A 0.000, B 0.000, C 0.000 }
gfCNCPoint5[20837] = {X 323.4682, Y 100.6004, Z -7.1667, A 0.000, B 0.000, C 0.000 }
gfCNCPoint5[20838] = {X 320.6876, Y 99.7923, Z -7.1667, A 0.000, B 0.000, C 0.000 }
gfCNCPoint5[20839] = {X 317.9740, Y 98.7819, Z -7.1667, A 0.000, B 0.000, C 0.000 }
gfCNCPoint5[20840] = {X 316.4793, Y 98.0924, Z -7.1667, A 0.000, B 0.000, C 0.000 }
gfCNCPoint5[20841] = {X 315.0474, Y 97.2803, Z -7.1667, A 0.000, B 0.000, C 0.000 }
gfCNCPoint5[20842] = {X 313.6883, Y 96.3515, Z -7.1667, A 0.000, B 0.000, C 0.000 }
gfCNCPoint5[20843] = {X 312.4117, Y 95.3123, Z -7.1667, A 0.000, B 0.000, C 0.000 }
gfCNCPoint5[20844] = {X 311.4281, Y 94.3336, Z -7.1667, A 0.000, B 0.000, C 0.000 }
gfCNCPoint5[20845] = {X 310.5673, Y 93.2453, Z -7.1667, A 0.000, B 0.000, C 0.000 }
gfCNCPoint5[20846] = {X 309.8416, Y 92.0626, Z -7.1667, A 0.000, B 0.000, C 0.000 }
gfCNCPoint5[20847] = {X 309.2611, Y 90.8024, Z -7.1667, A 0.000, B 0.000, C 0.000 }
gfCNCPoint5[20848] = {X 308.8340, Y 89.4822, Z -7.1667, A 0.000, B 0.000, C 0.000 }
gfCNCPoint5[20849] = {X 308.4948, Y 87.8792, Z -7.1667, A 0.000, B 0.000, C 0.000 }
gfCNCPoint5[20850] = {X 308.2945, Y 86.2530, Z -7.1667, A 0.000, B 0.000, C 0.000 }
gfCNCPoint5[20851] = {X 308.2344, Y 84.6156, Z -7.1667, A 0.000, B 0.000, C 0.000 }
gfCNCPoint5[20852] = {X 308.2356, Y 62.9981, Z -7.1667, A 0.000, B 0.000, C 0.000 }
gfCNCPoint5[20853] = {X 307.3941, Y 62.8330, Z -7.1667, A 0.000, B 0.000, C 0.000 }
gfCNCPoint5[20854] = {X 306.6057, Y 62.4956, Z -7.1667, A 0.000, B 0.000, C 0.000 }
gfCNCPoint5[20855] = {X 305.9052, Y 62.0008, Z -7.1667, A 0.000, B 0.000, C 0.000 }
gfCNCPoint5[20856] = {X 305.3237, Y 61.3706, Z -7.1667, A 0.000, B 0.000, C 0.000 }
gfCNCPoint5[20857] = {X 304.8866, Y 60.6327, Z -7.1667, A 0.000, B 0.000, C 0.000 }
gfCNCPoint5[20858] = {X 304.6135, Y 59.8198, Z -7.1667, A 0.000, B 0.000, C 0.000 }
gfCNCPoint5[20859] = {X 304.5164, Y 58.9678, Z -7.1667, A 0.000, B 0.000, C 0.000 }
gfCNCPoint5[20860] = {X 304.5162, Y 58.0000, Z -7.1667, A 0.000, B 0.000, C 0.000 }
gfCNCPoint5[20861] = {X 304.6185, Y 57.0921, Z -7.1667, A 0.000, B 0.000, C 0.000 }
gfCNCPoint5[20862] = {X 304.9203, Y 56.2298, Z -7.1667, A 0.000, B 0.000, C 0.000 }
gfCNCPoint5[20863] = {X 305.4064, Y 55.4562, Z -7.1667, A 0.000, B 0.000, C 0.000 }
gfCNCPoint5[20864] = {X 306.0524, Y 54.8101, Z -7.1667, A 0.000, B 0.000, C 0.000 }
gfCNCPoint5[20865] = {X 306.8260, Y 54.3240, Z -7.1667, A 0.000, B 0.000, C 0.000 }
gfCNCPoint5[20866] = {X 307.6883, Y 54.0223, Z -7.1667, A 0.000, B 0.000, C 0.000 }
gfCNCPoint5[20867] = {X 308.5962, Y 53.9200, Z -7.1667, A 0.000, B 0.000, C 0.000 }
gfCNCPoint5[20868] = {X 324.3107, Y 53.9200, Z -7.1667, A 0.000, B 0.000, C 0.000 }
gfCNCPoint5[20869] = {X 325.2186, Y 54.0223, Z -7.1667, A 0.000, B 0.000, C 0.000 }
gfCNCPoint5[20870] = {X 326.0809, Y 54.3240, Z -7.1667, A 0.000, B 0.000, C 0.000 }
gfCNCPoint5[20871] = {X 326.8545, Y 54.8101, Z -7.1667, A 0.000, B 0.000, C 0.000 }
gfCNCPoint5[20872] = {X 327.5006, Y 55.4562, Z -7.1667, A 0.000, B 0.000, C 0.000 }
gfCNCPoint5[20873] = {X 327.9866, Y 56.2298, Z -7.1667, A 0.000, B 0.000, C 0.000 }
gfCNCPoint5[20874] = {X 328.2884, Y 57.0921, Z -7.1667, A 0.000, B 0.000, C 0.000 }
gfCNCPoint5[20875] = {X 328.3907, Y 58.0000, Z -7.1667, A 0.000, B 0.000, C 0.000 }
gfCNCPoint5[20876] = {X 328.3907, Y 58.9345, Z -7.1667, A 0.000, B 0.000, C 0.000 }
gfCNCPoint5[20877] = {X 328.2959, Y 59.7915, Z -7.1667, A 0.000, B 0.000, C 0.000 }
gfCNCPoint5[20878] = {X 328.0247, Y 60.6099, Z -7.1667, A 0.000, B 0.000, C 0.000 }
gfCNCPoint5[20879] = {X 327.5891, Y 61.3539, Z -7.1667, A 0.000, B 0.000, C 0.000 }
gfCNCPoint5[20880] = {X 327.0080, Y 61.9908, Z -7.1667, A 0.000, B 0.000, C 0.000 }
gfCNCPoint5[20881] = {X 326.3071, Y 62.4928, Z -7.1667, A 0.000, B 0.000, C 0.000 }
gfCNCPoint5[20882] = {X 325.5170, Y 62.8378, Z -7.1667, A 0.000, B 0.000, C 0.000 }
gfCNCPoint5[20883] = {X 324.6723, Y 63.0107, Z -7.1667, A 0.000, B 0.000, C 0.000 }
gfCNCPoint5[20884] = {X 324.6742, Y 83.2308, Z -7.1667, A 0.000, B 0.000, C 0.000 }
gfCNCPoint5[20885] = {X 324.6878, Y 84.6156, Z -7.1667, A 0.000, B 0.000, C 0.000 }
gfCNCPoint5[20886] = {X 324.7695, Y 85.8992, Z -7.1667, A 0.000, B 0.000, C 0.000 }
gfCNCPoint5[20887] = {X 325.0029, Y 87.1641, Z -7.1667, A 0.000, B 0.000, C 0.000 }
gfCNCPoint5[20888] = {X 325.5046, Y 87.6526, Z -7.1667, A 0.000, B 0.000, C 0.000 }
gfCNCPoint5[20889] = {X 326.1101, Y 88.0045, Z -7.1667, A 0.000, B 0.000, C 0.000 }
gfCNCPoint5[20890] = {X 327.9147, Y 88.7256, Z -7.1667, A 0.000, B 0.000, C 0.000 }
gfCNCPoint5[20891] = {X 329.7927, Y 89.2253, Z -7.1667, A 0.000, B 0.000, C 0.000 }
gfCNCPoint5[20892] = {X 332.8903, Y 89.7809, Z -7.1667, A 0.000, B 0.000, C 0.000 }
gfCNCPoint5[20893] = {X 336.0160, Y 90.1468, Z -7.1667, A 0.000, B 0.000, C 0.000 }
gfCNCPoint5[20894] = {X 340.3936, Y 90.4416, Z -7.1667, A 0.000, B 0.000, C 0.000 }
gfCNCPoint5[20895] = {X 344.7784, Y 90.5957, Z -7.1667, A 0.000, B 0.000, C 0.000 }
gfCNCPoint5[20896] = {X 349.1659, Y 90.6090, Z -7.1667, A 0.000, B 0.000, C 0.000 }
gfCNCPoint5[20897] = {X 353.3251, Y 90.5404, Z -7.1667, A 0.000, B 0.000, C 0.000 }
gfCNCPoint5[20898] = {X 357.4791, Y 90.3210, Z -7.1667, A 0.000, B 0.000, C 0.000 }
gfCNCPoint5[20899] = {X 361.6224, Y 89.9509, Z -7.1667, A 0.000, B 0.000, C 0.000 }
gfCNCPoint5[20900] = {X 363.7169, Y 89.6620, Z -7.1667, A 0.000, B 0.000, C 0.000 }
gfCNCPoint5[20901] = {X 365.7921, Y 89.2575, Z -7.1667, A 0.000, B 0.000, C 0.000 }
gfCNCPoint5[20902] = {X 367.8417, Y 88.7386, Z -7.1667, A 0.000, B 0.000, C 0.000 }
gfCNCPoint5[20903] = {X 368.7991, Y 88.4170, Z -7.1667, A 0.000, B 0.000, C 0.000 }
gfCNCPoint5[20904] = {X 369.7142, Y 87.9897, Z -7.1667, A 0.000, B 0.000, C 0.000 }
gfCNCPoint5[20905] = {X 370.5755, Y 87.4622, Z -7.1667, A 0.000, B 0.000, C 0.000 }
gfCNCPoint5[20906] = {X 370.7901, Y 87.2387, Z -7.1667, A 0.000, B 0.000, C 0.000 }
gfCNCPoint5[20907] = {X 370.9008, Y 86.9492, Z -7.1667, A 0.000, B 0.000, C 0.000 }
gfCNCPoint5[20908] = {X 371.0944, Y 85.3944, Z -7.1667, A 0.000, B 0.000, C 0.000 }
gfCNCPoint5[20909] = {X 371.1591, Y 83.8288, Z -7.1667, A 0.000, B 0.000, C 0.000 }
gfCNCPoint5[20910] = {X 371.1600, Y 62.9982, Z -7.1667, A 0.000, B 0.000, C 0.000 }
gfCNCPoint5[20911] = {X 371.0234, Y 62.9838, Z -7.1667, A 0.000, B 0.000, C 0.000 }
gfCNCPoint5[20912] = {X 370.8874, Y 62.9648, Z -7.1667, A 0.000, B 0.000, C 0.000 }
gfCNCPoint5[20913] = {X 369.9681, Y 62.7077, Z -7.1667, A 0.000, B 0.000, C 0.000 }
gfCNCPoint5[20914] = {X 369.1337, Y 62.2440, Z -7.1667, A 0.000, B 0.000, C 0.000 }
gfCNCPoint5[20915] = {X 368.4299, Y 61.5991, Z -7.1667, A 0.000, B 0.000, C 0.000 }
gfCNCPoint5[20916] = {X 367.8952, Y 60.8083, Z -7.1667, A 0.000, B 0.000, C 0.000 }
gfCNCPoint5[20917] = {X 367.5589, Y 59.9149, Z -7.1667, A 0.000, B 0.000, C 0.000 }
gfCNCPoint5[20918] = {X 367.4394, Y 58.9678, Z -7.1667, A 0.000, B 0.000, C 0.000 }
gfCNCPoint5[20919] = {X 367.4393, Y 58.0000, Z -7.1667, A 0.000, B 0.000, C 0.000 }
gfCNCPoint5[20920] = {X 367.5416, Y 57.0921, Z -7.1667, A 0.000, B 0.000, C 0.000 }
gfCNCPoint5[20921] = {X 367.8433, Y 56.2298, Z -7.1667, A 0.000, B 0.000, C 0.000 }
gfCNCPoint5[20922] = {X 368.3294, Y 55.4562, Z -7.1667, A 0.000, B 0.000, C 0.000 }
gfCNCPoint5[20923] = {X 368.9754, Y 54.8101, Z -7.1667, A 0.000, B 0.000, C 0.000 }
gfCNCPoint5[20924] = {X 369.7490, Y 54.3240, Z -7.1667, A 0.000, B 0.000, C 0.000 }
gfCNCPoint5[20925] = {X 370.6114, Y 54.0223, Z -7.1667, A 0.000, B 0.000, C 0.000 }
gfCNCPoint5[20926] = {X 371.5193, Y 53.9200, Z -7.1667, A 0.000, B 0.000, C 0.000 }
gfCNCPoint5[20927] = {X 388.0597, Y 53.9200, Z -7.1667, A 0.000, B 0.000, C 0.000 }
gfCNCPoint5[20928] = {X 388.9676, Y 54.0223, Z -7.1667, A 0.000, B 0.000, C 0.000 }
gfCNCPoint5[20929] = {X 389.8299, Y 54.3240, Z -7.1667, A 0.000, B 0.000, C 0.000 }
gfCNCPoint5[20930] = {X 390.6035, Y 54.8101, Z -7.1667, A 0.000, B 0.000, C 0.000 }
gfCNCPoint5[20931] = {X 391.2496, Y 55.4562, Z -7.1667, A 0.000, B 0.000, C 0.000 }
gfCNCPoint5[20932] = {X 391.7356, Y 56.2298, Z -7.1667, A 0.000, B 0.000, C 0.000 }
gfCNCPoint5[20933] = {X 392.0374, Y 57.0921, Z -7.1667, A 0.000, B 0.000, C 0.000 }
gfCNCPoint5[20934] = {X 392.1397, Y 58.0000, Z -7.1667, A 0.000, B 0.000, C 0.000 }
gfCNCPoint5[20935] = {X 392.1397, Y 58.9342, Z -7.1667, A 0.000, B 0.000, C 0.000 }
gfCNCPoint5[20936] = {X 392.0343, Y 59.8555, Z -7.1667, A 0.000, B 0.000, C 0.000 }
gfCNCPoint5[20937] = {X 391.7235, Y 60.7293, Z -7.1667, A 0.000, B 0.000, C 0.000 }
gfCNCPoint5[20938] = {X 391.1914, Y 61.5503, Z -7.1667, A 0.000, B 0.000, C 0.000 }
gfCNCPoint5[20939] = {X 390.4800, Y 62.2219, Z -7.1667, A 0.000, B 0.000, C 0.000 }
gfCNCPoint5[20940] = {X 389.6298, Y 62.7061, Z -7.1667, A 0.000, B 0.000, C 0.000 }
gfCNCPoint5[20941] = {X 388.6892, Y 62.9753, Z -7.1667, A 0.000, B 0.000, C 0.000 }
gfCNCPoint5[20942] = {X 388.5560, Y 62.9945, Z -7.1667, A 0.000, B 0.000, C 0.000 }
gfCNCPoint5[20943] = {X 388.4222, Y 63.0093, Z -7.1667, A 0.000, B 0.000, C 0.000 }
gfCNCPoint5[20944] = {X 388.4200, Y 63.1547, Z -7.1667, A 0.000, B 0.000, C 0.000 }
gfCNCPoint5[20945] = {X 388.4179, Y 84.6157, Z -7.1667, A 0.000, B 0.000, C 0.000 }
gfCNCPoint5[20946] = {X 388.3588, Y 86.2534, Z -7.1667, A 0.000, B 0.000, C 0.000 }
gfCNCPoint5[20947] = {X 388.1571, Y 87.8797, Z -7.1667, A 0.000, B 0.000, C 0.000 }
gfCNCPoint5[20948] = {X 387.8142, Y 89.4822, Z -7.1667, A 0.000, B 0.000, C 0.000 }
gfCNCPoint5[20949] = {X 387.2924, Y 91.0374, Z -7.1667, A 0.000, B 0.000, C 0.000 }
gfCNCPoint5[20950] = {X 386.5579, Y 92.5042, Z -7.1667, A 0.000, B 0.000, C 0.000 }
gfCNCPoint5[20951] = {X 385.6251, Y 93.8535, Z -7.1667, A 0.000, B 0.000, C 0.000 }
gfCNCPoint5[20952] = {X 384.5124, Y 95.0589, Z -7.1667, A 0.000, B 0.000, C 0.000 }
gfCNCPoint5[20953] = {X 383.0173, Y 96.3190, Z -7.1667, A 0.000, B 0.000, C 0.000 }
gfCNCPoint5[20954] = {X 381.3968, Y 97.4131, Z -7.1667, A 0.000, B 0.000, C 0.000 }
gfCNCPoint5[20955] = {X 379.6693, Y 98.3289, Z -7.1667, A 0.000, B 0.000, C 0.000 }
gfCNCPoint5[20956] = {X 377.4137, Y 99.2772, Z -7.1667, A 0.000, B 0.000, C 0.000 }
gfCNCPoint5[20957] = {X 375.0960, Y 100.0619, Z -7.1667, A 0.000, B 0.000, C 0.000 }
gfCNCPoint5[20958] = {X 372.7282, Y 100.6790, Z -7.1667, A 0.000, B 0.000, C 0.000 }
gfCNCPoint5[20959] = {X 368.8292, Y 101.4299, Z -7.1667, A 0.000, B 0.000, C 0.000 }
gfCNCPoint5[20960] = {X 364.8980, Y 101.9885, Z -7.1667, A 0.000, B 0.000, C 0.000 }
gfCNCPoint5[20961] = {X 360.9441, Y 102.3534, Z -7.1667, A 0.000, B 0.000, C 0.000 }
gfCNCPoint5[20962] = {X 357.0919, Y 102.5780, Z -7.1667, A 0.000, B 0.000, C 0.000 }
gfCNCPoint5[20963] = {X 353.2360, Y 102.7232, Z -7.1667, A 0.000, B 0.000, C 0.000 }
gfCNCPoint5[20964] = {X 353.3452, Y 106.7217, Z -7.1667, A 0.000, B 0.000, C 0.000 }
gfCNCPoint5[20965] = {X 353.2338, Y 102.6432, Z -7.1667, A 0.000, B 0.000, C 0.000 }
gfCNCPoint5[20966] = {X 348.1835, Y 102.7129, Z -7.1667, A 0.000, B 0.000, C 0.000 }
gfCNCPoint5[20967] = {X 343.1333, Y 102.6463, Z -7.1667, A 0.000, B 0.000, C 0.000 }
gfCNCPoint5[20968] = {X 338.0866, Y 102.4432, Z -7.1667, A 0.000, B 0.000, C 0.000 }
gfCNCPoint5[20969] = {X 334.1453, Y 102.1672, Z -7.1667, A 0.000, B 0.000, C 0.000 }
gfCNCPoint5[20970] = {X 330.2189, Y 101.7268, Z -7.1667, A 0.000, B 0.000, C 0.000 }
gfCNCPoint5[20971] = {X 326.3144, Y 101.1228, Z -7.1667, A 0.000, B 0.000, C 0.000 }
gfCNCPoint5[20972] = {X 323.4876, Y 100.5228, Z -7.1667, A 0.000, B 0.000, C 0.000 }
gfCNCPoint5[20973] = {X 320.7127, Y 99.7164, Z -7.1667, A 0.000, B 0.000, C 0.000 }
gfCNCPoint5[20974] = {X 318.0046, Y 98.7079, Z -7.1667, A 0.000, B 0.000, C 0.000 }
gfCNCPoint5[20975] = {X 316.5159, Y 98.0212, Z -7.1667, A 0.000, B 0.000, C 0.000 }
gfCNCPoint5[20976] = {X 315.0897, Y 97.2125, Z -7.1667, A 0.000, B 0.000, C 0.000 }
gfCNCPoint5[20977] = {X 313.7362, Y 96.2874, Z -7.1667, A 0.000, B 0.000, C 0.000 }
gfCNCPoint5[20978] = {X 312.4647, Y 95.2524, Z -7.1667, A 0.000, B 0.000, C 0.000 }
gfCNCPoint5[20979] = {X 311.4878, Y 94.2804, Z -7.1667, A 0.000, B 0.000, C 0.000 }
gfCNCPoint5[20980] = {X 310.6330, Y 93.1995, Z -7.1667, A 0.000, B 0.000, C 0.000 }
gfCNCPoint5[20981] = {X 309.9122, Y 92.0250, Z -7.1667, A 0.000, B 0.000, C 0.000 }
gfCNCPoint5[20982] = {X 309.3356, Y 90.7733, Z -7.1667, A 0.000, B 0.000, C 0.000 }
gfCNCPoint5[20983] = {X 308.9114, Y 89.4621, Z -7.1667, A 0.000, B 0.000, C 0.000 }
gfCNCPoint5[20984] = {X 308.5737, Y 87.8658, Z -7.1667, A 0.000, B 0.000, C 0.000 }
gfCNCPoint5[20985] = {X 308.3742, Y 86.2464, Z -7.1667, A 0.000, B 0.000, C 0.000 }
gfCNCPoint5[20986] = {X 308.3144, Y 84.6159, Z -7.1667, A 0.000, B 0.000, C 0.000 }
gfCNCPoint5[20987] = {X 308.3156, Y 62.9242, Z -7.1667, A 0.000, B 0.000, C 0.000 }
gfCNCPoint5[20988] = {X 307.4732, Y 62.7732, Z -7.1667, A 0.000, B 0.000, C 0.000 }
gfCNCPoint5[20989] = {X 306.6822, Y 62.4464, Z -7.1667, A 0.000, B 0.000, C 0.000 }
gfCNCPoint5[20990] = {X 305.9788, Y 61.9589, Z -7.1667, A 0.000, B 0.000, C 0.000 }
gfCNCPoint5[20991] = {X 305.3953, Y 61.3328, Z -7.1667, A 0.000, B 0.000, C 0.000 }
gfCNCPoint5[20992] = {X 304.9583, Y 60.5970, Z -7.1667, A 0.000, B 0.000, C 0.000 }
gfCNCPoint5[20993] = {X 304.6878, Y 59.7850, Z -7.1667, A 0.000, B 0.000, C 0.000 }
gfCNCPoint5[20994] = {X 304.5962, Y 58.9341, Z -7.1667, A 0.000, B 0.000, C 0.000 }
gfCNCPoint5[20995] = {X 304.5962, Y 58.0000, Z -7.1667, A 0.000, B 0.000, C 0.000 }
gfCNCPoint5[20996] = {X 304.6965, Y 57.1099, Z -7.1667, A 0.000, B 0.000, C 0.000 }
gfCNCPoint5[20997] = {X 304.9923, Y 56.2645, Z -7.1667, A 0.000, B 0.000, C 0.000 }
gfCNCPoint5[20998] = {X 305.4689, Y 55.5060, Z -7.1667, A 0.000, B 0.000, C 0.000 }
gfCNCPoint5[20999] = {X 306.1023, Y 54.8727, Z -7.1667, A 0.000, B 0.000, C 0.000 }
gfCNCPoint5[21000] = {X 306.8607, Y 54.3961, Z -7.1667, A 0.000, B 0.000, C 0.000 }
gfCNCPoint5[21001] = {X 307.7061, Y 54.1003, Z -7.1667, A 0.000, B 0.000, C 0.000 }
gfCNCPoint5[21002] = {X 308.5962, Y 54.0000, Z -7.1667, A 0.000, B 0.000, C 0.000 }
gfCNCPoint5[21003] = {X 324.3107, Y 54.0000, Z -7.1667, A 0.000, B 0.000, C 0.000 }
gfCNCPoint5[21004] = {X 325.2008, Y 54.1003, Z -7.1667, A 0.000, B 0.000, C 0.000 }
gfCNCPoint5[21005] = {X 326.0462, Y 54.3961, Z -7.1667, A 0.000, B 0.000, C 0.000 }
gfCNCPoint5[21006] = {X 326.8046, Y 54.8727, Z -7.1667, A 0.000, B 0.000, C 0.000 }
gfCNCPoint5[21007] = {X 327.4380, Y 55.5060, Z -7.1667, A 0.000, B 0.000, C 0.000 }
gfCNCPoint5[21008] = {X 327.9146, Y 56.2645, Z -7.1667, A 0.000, B 0.000, C 0.000 }
gfCNCPoint5[21009] = {X 328.2104, Y 57.1099, Z -7.1667, A 0.000, B 0.000, C 0.000 }
gfCNCPoint5[21010] = {X 328.3107, Y 58.0000, Z -7.1667, A 0.000, B 0.000, C 0.000 }
gfCNCPoint5[21011] = {X 328.3107, Y 58.9341, Z -7.1667, A 0.000, B 0.000, C 0.000 }
gfCNCPoint5[21012] = {X 328.2155, Y 59.7845, Z -7.1667, A 0.000, B 0.000, C 0.000 }
gfCNCPoint5[21013] = {X 327.9433, Y 60.5958, Z -7.1667, A 0.000, B 0.000, C 0.000 }
gfCNCPoint5[21014] = {X 327.5061, Y 61.3314, Z -7.1667, A 0.000, B 0.000, C 0.000 }
gfCNCPoint5[21015] = {X 326.9238, Y 61.9584, Z -7.1667, A 0.000, B 0.000, C 0.000 }
gfCNCPoint5[21016] = {X 326.2224, Y 62.4486, Z -7.1667, A 0.000, B 0.000, C 0.000 }
gfCNCPoint5[21017] = {X 325.4334, Y 62.7799, Z -7.1667, A 0.000, B 0.000, C 0.000 }
gfCNCPoint5[21018] = {X 324.5923, Y 62.9375, Z -7.1667, A 0.000, B 0.000, C 0.000 }
gfCNCPoint5[21019] = {X 324.5942, Y 83.2313, Z -7.1667, A 0.000, B 0.000, C 0.000 }
gfCNCPoint5[21020] = {X 324.6078, Y 84.6159, Z -7.1667, A 0.000, B 0.000, C 0.000 }
gfCNCPoint5[21021] = {X 324.6912, Y 85.9177, Z -7.1667, A 0.000, B 0.000, C 0.000 }
gfCNCPoint5[21022] = {X 324.9294, Y 87.2003, Z -7.1667, A 0.000, B 0.000, C 0.000 }
gfCNCPoint5[21023] = {X 325.4486, Y 87.7105, Z -7.1667, A 0.000, B 0.000, C 0.000 }
gfCNCPoint5[21024] = {X 326.0773, Y 88.0775, Z -7.1667, A 0.000, B 0.000, C 0.000 }
gfCNCPoint5[21025] = {X 327.8902, Y 88.8018, Z -7.1667, A 0.000, B 0.000, C 0.000 }
gfCNCPoint5[21026] = {X 329.7768, Y 89.3037, Z -7.1667, A 0.000, B 0.000, C 0.000 }
gfCNCPoint5[21027] = {X 332.8789, Y 89.8601, Z -7.1667, A 0.000, B 0.000, C 0.000 }
gfCNCPoint5[21028] = {X 336.0092, Y 90.2265, Z -7.1667, A 0.000, B 0.000, C 0.000 }
gfCNCPoint5[21029] = {X 340.3892, Y 90.5215, Z -7.1667, A 0.000, B 0.000, C 0.000 }
gfCNCPoint5[21030] = {X 344.7764, Y 90.6757, Z -7.1667, A 0.000, B 0.000, C 0.000 }
gfCNCPoint5[21031] = {X 349.1664, Y 90.6890, Z -7.1667, A 0.000, B 0.000, C 0.000 }
gfCNCPoint5[21032] = {X 353.3283, Y 90.6204, Z -7.1667, A 0.000, B 0.000, C 0.000 }
gfCNCPoint5[21033] = {X 357.4851, Y 90.4008, Z -7.1667, A 0.000, B 0.000, C 0.000 }
gfCNCPoint5[21034] = {X 361.6311, Y 90.0305, Z -7.1667, A 0.000, B 0.000, C 0.000 }
gfCNCPoint5[21035] = {X 363.7299, Y 89.7410, Z -7.1667, A 0.000, B 0.000, C 0.000 }
gfCNCPoint5[21036] = {X 365.8095, Y 89.3356, Z -7.1667, A 0.000, B 0.000, C 0.000 }
gfCNCPoint5[21037] = {X 367.8634, Y 88.8155, Z -7.1667, A 0.000, B 0.000, C 0.000 }
gfCNCPoint5[21038] = {X 368.8292, Y 88.4911, Z -7.1667, A 0.000, B 0.000, C 0.000 }
gfCNCPoint5[21039] = {X 369.7523, Y 88.0601, Z -7.1667, A 0.000, B 0.000, C 0.000 }
gfCNCPoint5[21040] = {X 370.6211, Y 87.5280, Z -7.1667, A 0.000, B 0.000, C 0.000 }
gfCNCPoint5[21041] = {X 370.8577, Y 87.2815, Z -7.1667, A 0.000, B 0.000, C 0.000 }
gfCNCPoint5[21042] = {X 370.9797, Y 86.9624, Z -7.1667, A 0.000, B 0.000, C 0.000 }
gfCNCPoint5[21043] = {X 371.1742, Y 85.4010, Z -7.1667, A 0.000, B 0.000, C 0.000 }
gfCNCPoint5[21044] = {X 371.2391, Y 83.8288, Z -7.1667, A 0.000, B 0.000, C 0.000 }
gfCNCPoint5[21045] = {X 371.2379, Y 63.0399, Z -7.1667, A 0.000, B 0.000, C 0.000 }
gfCNCPoint5[21046] = {X 371.2440, Y 62.9246, Z -7.1667, A 0.000, B 0.000, C 0.000 }
gfCNCPoint5[21047] = {X 371.0715, Y 62.9089, Z -7.1667, A 0.000, B 0.000, C 0.000 }
gfCNCPoint5[21048] = {X 370.8998, Y 62.8858, Z -7.1667, A 0.000, B 0.000, C 0.000 }
gfCNCPoint5[21049] = {X 369.9934, Y 62.6316, Z -7.1667, A 0.000, B 0.000, C 0.000 }
gfCNCPoint5[21050] = {X 369.1716, Y 62.1726, Z -7.1667, A 0.000, B 0.000, C 0.000 }
gfCNCPoint5[21051] = {X 368.4797, Y 61.5343, Z -7.1667, A 0.000, B 0.000, C 0.000 }
gfCNCPoint5[21052] = {X 367.9562, Y 60.7519, Z -7.1667, A 0.000, B 0.000, C 0.000 }
gfCNCPoint5[21053] = {X 367.6300, Y 59.8689, Z -7.1667, A 0.000, B 0.000, C 0.000 }
gfCNCPoint5[21054] = {X 367.5193, Y 58.9341, Z -7.1667, A 0.000, B 0.000, C 0.000 }
gfCNCPoint5[21055] = {X 367.5193, Y 58.0000, Z -7.1667, A 0.000, B 0.000, C 0.000 }
gfCNCPoint5[21056] = {X 367.6196, Y 57.1099, Z -7.1667, A 0.000, B 0.000, C 0.000 }
gfCNCPoint5[21057] = {X 367.9154, Y 56.2645, Z -7.1667, A 0.000, B 0.000, C 0.000 }
gfCNCPoint5[21058] = {X 368.3920, Y 55.5060, Z -7.1667, A 0.000, B 0.000, C 0.000 }
gfCNCPoint5[21059] = {X 369.0253, Y 54.8727, Z -7.1667, A 0.000, B 0.000, C 0.000 }
gfCNCPoint5[21060] = {X 369.7837, Y 54.3961, Z -7.1667, A 0.000, B 0.000, C 0.000 }
gfCNCPoint5[21061] = {X 370.6292, Y 54.1003, Z -7.1667, A 0.000, B 0.000, C 0.000 }
gfCNCPoint5[21062] = {X 371.5193, Y 54.0000, Z -7.1667, A 0.000, B 0.000, C 0.000 }
gfCNCPoint5[21063] = {X 388.0597, Y 54.0000, Z -7.1667, A 0.000, B 0.000, C 0.000 }
gfCNCPoint5[21064] = {X 388.9498, Y 54.1003, Z -7.1667, A 0.000, B 0.000, C 0.000 }
gfCNCPoint5[21065] = {X 389.7952, Y 54.3961, Z -7.1667, A 0.000, B 0.000, C 0.000 }
gfCNCPoint5[21066] = {X 390.5536, Y 54.8727, Z -7.1667, A 0.000, B 0.000, C 0.000 }
gfCNCPoint5[21067] = {X 391.1870, Y 55.5060, Z -7.1667, A 0.000, B 0.000, C 0.000 }
gfCNCPoint5[21068] = {X 391.6636, Y 56.2645, Z -7.1667, A 0.000, B 0.000, C 0.000 }
gfCNCPoint5[21069] = {X 391.9594, Y 57.1099, Z -7.1667, A 0.000, B 0.000, C 0.000 }
gfCNCPoint5[21070] = {X 392.0597, Y 58.0000, Z -7.1667, A 0.000, B 0.000, C 0.000 }
gfCNCPoint5[21071] = {X 392.0595, Y 58.9671, Z -7.1667, A 0.000, B 0.000, C 0.000 }
gfCNCPoint5[21072] = {X 391.9526, Y 59.8535, Z -7.1667, A 0.000, B 0.000, C 0.000 }
gfCNCPoint5[21073] = {X 391.6517, Y 60.6941, Z -7.1667, A 0.000, B 0.000, C 0.000 }
gfCNCPoint5[21074] = {X 391.1299, Y 61.4991, Z -7.1667, A 0.000, B 0.000, C 0.000 }
gfCNCPoint5[21075] = {X 390.4324, Y 62.1576, Z -7.1667, A 0.000, B 0.000, C 0.000 }
gfCNCPoint5[21076] = {X 389.5988, Y 62.6324, Z -7.1667, A 0.000, B 0.000, C 0.000 }
gfCNCPoint5[21077] = {X 388.6765, Y 62.8963, Z -7.1667, A 0.000, B 0.000, C 0.000 }
gfCNCPoint5[21078] = {X 388.5103, Y 62.9195, Z -7.1667, A 0.000, B 0.000, C 0.000 }
gfCNCPoint5[21079] = {X 388.3432, Y 62.9357, Z -7.1667, A 0.000, B 0.000, C 0.000 }
gfCNCPoint5[21080] = {X 388.3400, Y 63.1540, Z -7.1667, A 0.000, B 0.000, C 0.000 }
gfCNCPoint5[21081] = {X 388.3400, Y 83.9236, Z -7.1667, A 0.000, B 0.000, C 0.000 }
gfCNCPoint5[21082] = {X 388.3379, Y 84.6159, Z -7.1667, A 0.000, B 0.000, C 0.000 }
gfCNCPoint5[21083] = {X 388.2791, Y 86.2468, Z -7.1667, A 0.000, B 0.000, C 0.000 }
gfCNCPoint5[21084] = {X 388.0782, Y 87.8663, Z -7.1667, A 0.000, B 0.000, C 0.000 }
gfCNCPoint5[21085] = {X 387.7367, Y 89.4621, Z -7.1667, A 0.000, B 0.000, C 0.000 }
gfCNCPoint5[21086] = {X 387.2185, Y 91.0067, Z -7.1667, A 0.000, B 0.000, C 0.000 }
gfCNCPoint5[21087] = {X 386.4890, Y 92.4634, Z -7.1667, A 0.000, B 0.000, C 0.000 }
gfCNCPoint5[21088] = {X 385.5626, Y 93.8035, Z -7.1667, A 0.000, B 0.000, C 0.000 }
gfCNCPoint5[21089] = {X 384.4576, Y 95.0007, Z -7.1667, A 0.000, B 0.000, C 0.000 }
gfCNCPoint5[21090] = {X 382.9690, Y 96.2552, Z -7.1667, A 0.000, B 0.000, C 0.000 }
gfCNCPoint5[21091] = {X 381.3556, Y 97.3445, Z -7.1667, A 0.000, B 0.000, C 0.000 }
gfCNCPoint5[21092] = {X 379.6357, Y 98.2563, Z -7.1667, A 0.000, B 0.000, C 0.000 }
gfCNCPoint5[21093] = {X 377.3853, Y 99.2024, Z -7.1667, A 0.000, B 0.000, C 0.000 }
gfCNCPoint5[21094] = {X 375.0731, Y 99.9852, Z -7.1667, A 0.000, B 0.000, C 0.000 }
gfCNCPoint5[21095] = {X 372.7108, Y 100.6009, Z -7.1667, A 0.000, B 0.000, C 0.000 }
gfCNCPoint5[21096] = {X 368.8157, Y 101.3510, Z -7.1667, A 0.000, B 0.000, C 0.000 }
gfCNCPoint5[21097] = {X 364.8885, Y 101.9090, Z -7.1667, A 0.000, B 0.000, C 0.000 }
gfCNCPoint5[21098] = {X 360.9386, Y 102.2735, Z -7.1667, A 0.000, B 0.000, C 0.000 }
gfCNCPoint5[21099] = {X 357.0881, Y 102.4981, Z -7.1667, A 0.000, B 0.000, C 0.000 }
gfCNCPoint5[21100] = {X 353.2338, Y 102.6432, Z -7.1667, A 0.000, B 0.000, C 0.000 }
gfCNCPoint5[21101] = {X 353.3452, Y 106.7217, Z -7.1667, A 0.000, B 0.000, C 0.000 }
gfCNCPoint5[21102] = {X 353.3452, Y 106.7217, Z -4.1667, A 0.000, B 0.000, C 0.000 }
gfCNCPoint5[21103] = {X 353.3452, Y 106.7217, Z 11.0000, A 0.000, B 0.000, C 0.000 }
gfCNCPoint5[21104] = {X 411.5984, Y 79.5922, Z 11.0000, A 0.000, B 0.000, C 0.000 }
gfCNCPoint5[21105] = {X 411.5984, Y 79.5922, Z -4.1667, A 0.000, B 0.000, C 0.000 }
gfCNCPoint5[21106] = {X 411.5984, Y 79.5922, Z -7.1667, A 0.000, B 0.000, C 0.000 }
gfCNCPoint5[21107] = {X 413.7986, Y 83.0281, Z -7.1667, A 0.000, B 0.000, C 0.000 }
gfCNCPoint5[21108] = {X 428.0535, Y 73.8996, Z -7.1667, A 0.000, B 0.000, C 0.000 }
gfCNCPoint5[21109] = {X 403.7555, Y 64.3669, Z -7.1667, A 0.000, B 0.000, C 0.000 }
gfCNCPoint5[21110] = {X 402.0595, Y 63.8055, Z -7.1667, A 0.000, B 0.000, C 0.000 }
gfCNCPoint5[21111] = {X 400.3122, Y 63.4330, Z -7.1667, A 0.000, B 0.000, C 0.000 }
gfCNCPoint5[21112] = {X 398.5347, Y 63.2540, Z -7.1667, A 0.000, B 0.000, C 0.000 }
gfCNCPoint5[21113] = {X 397.5822, Y 63.1425, Z -7.1667, A 0.000, B 0.000, C 0.000 }
gfCNCPoint5[21114] = {X 396.6777, Y 62.8235, Z -7.1667, A 0.000, B 0.000, C 0.000 }
gfCNCPoint5[21115] = {X 395.8659, Y 62.3129, Z -7.1667, A 0.000, B 0.000, C 0.000 }
gfCNCPoint5[21116] = {X 395.1868, Y 61.6358, Z -7.1667, A 0.000, B 0.000, C 0.000 }
gfCNCPoint5[21117] = {X 394.6738, Y 60.8255, Z -7.1667, A 0.000, B 0.000, C 0.000 }
gfCNCPoint5[21118] = {X 394.3522, Y 59.9219, Z -7.1667, A 0.000, B 0.000, C 0.000 }
gfCNCPoint5[21119] = {X 394.2379, Y 58.9697, Z -7.1667, A 0.000, B 0.000, C 0.000 }
gfCNCPoint5[21120] = {X 394.2377, Y 58.0000, Z -7.1667, A 0.000, B 0.000, C 0.000 }
gfCNCPoint5[21121] = {X 394.3460, Y 57.0387, Z -7.1667, A 0.000, B 0.000, C 0.000 }
gfCNCPoint5[21122] = {X 394.6655, Y 56.1256, Z -7.1667, A 0.000, B 0.000, C 0.000 }
gfCNCPoint5[21123] = {X 395.1802, Y 55.3065, Z -7.1667, A 0.000, B 0.000, C 0.000 }
gfCNCPoint5[21124] = {X 395.8642, Y 54.6225, Z -7.1667, A 0.000, B 0.000, C 0.000 }
gfCNCPoint5[21125] = {X 396.6833, Y 54.1078, Z -7.1667, A 0.000, B 0.000, C 0.000 }
gfCNCPoint5[21126] = {X 397.5964, Y 53.7883, Z -7.1667, A 0.000, B 0.000, C 0.000 }
gfCNCPoint5[21127] = {X 398.5577, Y 53.6800, Z -7.1667, A 0.000, B 0.000, C 0.000 }
gfCNCPoint5[21128] = {X 419.4886, Y 53.6800, Z -7.1667, A 0.000, B 0.000, C 0.000 }
gfCNCPoint5[21129] = {X 420.4499, Y 53.7883, Z -7.1667, A 0.000, B 0.000, C 0.000 }
gfCNCPoint5[21130] = {X 421.3630, Y 54.1078, Z -7.1667, A 0.000, B 0.000, C 0.000 }
gfCNCPoint5[21131] = {X 422.1821, Y 54.6225, Z -7.1667, A 0.000, B 0.000, C 0.000 }
gfCNCPoint5[21132] = {X 422.8661, Y 55.3065, Z -7.1667, A 0.000, B 0.000, C 0.000 }
gfCNCPoint5[21133] = {X 423.3808, Y 56.1256, Z -7.1667, A 0.000, B 0.000, C 0.000 }
gfCNCPoint5[21134] = {X 423.7003, Y 57.0387, Z -7.1667, A 0.000, B 0.000, C 0.000 }
gfCNCPoint5[21135] = {X 423.8086, Y 58.0000, Z -7.1667, A 0.000, B 0.000, C 0.000 }
gfCNCPoint5[21136] = {X 423.8086, Y 58.2316, Z -7.1667, A 0.000, B 0.000, C 0.000 }
gfCNCPoint5[21137] = {X 429.6116, Y 60.4924, Z -7.1667, A 0.000, B 0.000, C 0.000 }
gfCNCPoint5[21138] = {X 457.8581, Y 71.6998, Z -7.1667, A 0.000, B 0.000, C 0.000 }
gfCNCPoint5[21139] = {X 457.8602, Y 63.2123, Z -7.1667, A 0.000, B 0.000, C 0.000 }
gfCNCPoint5[21140] = {X 457.0086, Y 63.0031, Z -7.1667, A 0.000, B 0.000, C 0.000 }
gfCNCPoint5[21141] = {X 456.2168, Y 62.6263, Z -7.1667, A 0.000, B 0.000, C 0.000 }
gfCNCPoint5[21142] = {X 455.5175, Y 62.0973, Z -7.1667, A 0.000, B 0.000, C 0.000 }
gfCNCPoint5[21143] = {X 454.9393, Y 61.4380, Z -7.1667, A 0.000, B 0.000, C 0.000 }
gfCNCPoint5[21144] = {X 454.5062, Y 60.6756, Z -7.1667, A 0.000, B 0.000, C 0.000 }
gfCNCPoint5[21145] = {X 454.2360, Y 59.8413, Z -7.1667, A 0.000, B 0.000, C 0.000 }
gfCNCPoint5[21146] = {X 454.1398, Y 58.9697, Z -7.1667, A 0.000, B 0.000, C 0.000 }
gfCNCPoint5[21147] = {X 454.1396, Y 58.0000, Z -7.1667, A 0.000, B 0.000, C 0.000 }
gfCNCPoint5[21148] = {X 454.2479, Y 57.0387, Z -7.1667, A 0.000, B 0.000, C 0.000 }
gfCNCPoint5[21149] = {X 454.5674, Y 56.1256, Z -7.1667, A 0.000, B 0.000, C 0.000 }
gfCNCPoint5[21150] = {X 455.0821, Y 55.3065, Z -7.1667, A 0.000, B 0.000, C 0.000 }
gfCNCPoint5[21151] = {X 455.7661, Y 54.6225, Z -7.1667, A 0.000, B 0.000, C 0.000 }
gfCNCPoint5[21152] = {X 456.5852, Y 54.1078, Z -7.1667, A 0.000, B 0.000, C 0.000 }
gfCNCPoint5[21153] = {X 457.4983, Y 53.7883, Z -7.1667, A 0.000, B 0.000, C 0.000 }
gfCNCPoint5[21154] = {X 458.4596, Y 53.6800, Z -7.1667, A 0.000, B 0.000, C 0.000 }
gfCNCPoint5[21155] = {X 475.0000, Y 53.6800, Z -7.1667, A 0.000, B 0.000, C 0.000 }
gfCNCPoint5[21156] = {X 475.9613, Y 53.7883, Z -7.1667, A 0.000, B 0.000, C 0.000 }
gfCNCPoint5[21157] = {X 476.8744, Y 54.1078, Z -7.1667, A 0.000, B 0.000, C 0.000 }
gfCNCPoint5[21158] = {X 477.6935, Y 54.6225, Z -7.1667, A 0.000, B 0.000, C 0.000 }
gfCNCPoint5[21159] = {X 478.3775, Y 55.3065, Z -7.1667, A 0.000, B 0.000, C 0.000 }
gfCNCPoint5[21160] = {X 478.8922, Y 56.1256, Z -7.1667, A 0.000, B 0.000, C 0.000 }
gfCNCPoint5[21161] = {X 479.2117, Y 57.0387, Z -7.1667, A 0.000, B 0.000, C 0.000 }
gfCNCPoint5[21162] = {X 479.3200, Y 58.0000, Z -7.1667, A 0.000, B 0.000, C 0.000 }
gfCNCPoint5[21163] = {X 479.3200, Y 58.9342, Z -7.1667, A 0.000, B 0.000, C 0.000 }
gfCNCPoint5[21164] = {X 479.2300, Y 59.8113, Z -7.1667, A 0.000, B 0.000, C 0.000 }
gfCNCPoint5[21165] = {X 478.9638, Y 60.6519, Z -7.1667, A 0.000, B 0.000, C 0.000 }
gfCNCPoint5[21166] = {X 478.5324, Y 61.4209, Z -7.1667, A 0.000, B 0.000, C 0.000 }
gfCNCPoint5[21167] = {X 477.9539, Y 62.0863, Z -7.1667, A 0.000, B 0.000, C 0.000 }
gfCNCPoint5[21168] = {X 477.2524, Y 62.6204, Z -7.1667, A 0.000, B 0.000, C 0.000 }
gfCNCPoint5[21169] = {X 476.4570, Y 63.0009, Z -7.1667, A 0.000, B 0.000, C 0.000 }
gfCNCPoint5[21170] = {X 475.6010, Y 63.2121, Z -7.1667, A 0.000, B 0.000, C 0.000 }
gfCNCPoint5[21171] = {X 475.6014, Y 92.7674, Z -7.1667, A 0.000, B 0.000, C 0.000 }
gfCNCPoint5[21172] = {X 475.9935, Y 92.8652, Z -7.1667, A 0.000, B 0.000, C 0.000 }
gfCNCPoint5[21173] = {X 476.3800, Y 92.9830, Z -7.1667, A 0.000, B 0.000, C 0.000 }
gfCNCPoint5[21174] = {X 477.1936, Y 93.3519, Z -7.1667, A 0.000, B 0.000, C 0.000 }
gfCNCPoint5[21175] = {X 477.9135, Y 93.8810, Z -7.1667, A 0.000, B 0.000, C 0.000 }
gfCNCPoint5[21176] = {X 478.5084, Y 94.5475, Z -7.1667, A 0.000, B 0.000, C 0.000 }
gfCNCPoint5[21177] = {X 478.9527, Y 95.3225, Z -7.1667, A 0.000, B 0.000, C 0.000 }
gfCNCPoint5[21178] = {X 479.2272, Y 96.1726, Z -7.1667, A 0.000, B 0.000, C 0.000 }
gfCNCPoint5[21179] = {X 479.3200, Y 97.0611, Z -7.1667, A 0.000, B 0.000, C 0.000 }
gfCNCPoint5[21180] = {X 479.3200, Y 98.0000, Z -7.1667, A 0.000, B 0.000, C 0.000 }
gfCNCPoint5[21181] = {X 479.2117, Y 98.9613, Z -7.1667, A 0.000, B 0.000, C 0.000 }
gfCNCPoint5[21182] = {X 478.8922, Y 99.8744, Z -7.1667, A 0.000, B 0.000, C 0.000 }
gfCNCPoint5[21183] = {X 478.3775, Y 100.6935, Z -7.1667, A 0.000, B 0.000, C 0.000 }
gfCNCPoint5[21184] = {X 477.6935, Y 101.3775, Z -7.1667, A 0.000, B 0.000, C 0.000 }
gfCNCPoint5[21185] = {X 476.8744, Y 101.8922, Z -7.1667, A 0.000, B 0.000, C 0.000 }
gfCNCPoint5[21186] = {X 475.9613, Y 102.2117, Z -7.1667, A 0.000, B 0.000, C 0.000 }
gfCNCPoint5[21187] = {X 475.0000, Y 102.3200, Z -7.1667, A 0.000, B 0.000, C 0.000 }
gfCNCPoint5[21188] = {X 458.4596, Y 102.3200, Z -7.1667, A 0.000, B 0.000, C 0.000 }
gfCNCPoint5[21189] = {X 457.4983, Y 102.2117, Z -7.1667, A 0.000, B 0.000, C 0.000 }
gfCNCPoint5[21190] = {X 456.5852, Y 101.8922, Z -7.1667, A 0.000, B 0.000, C 0.000 }
gfCNCPoint5[21191] = {X 455.7661, Y 101.3775, Z -7.1667, A 0.000, B 0.000, C 0.000 }
gfCNCPoint5[21192] = {X 455.0821, Y 100.6935, Z -7.1667, A 0.000, B 0.000, C 0.000 }
gfCNCPoint5[21193] = {X 454.5674, Y 99.8744, Z -7.1667, A 0.000, B 0.000, C 0.000 }
gfCNCPoint5[21194] = {X 454.2479, Y 98.9613, Z -7.1667, A 0.000, B 0.000, C 0.000 }
gfCNCPoint5[21195] = {X 454.1396, Y 98.0000, Z -7.1667, A 0.000, B 0.000, C 0.000 }
gfCNCPoint5[21196] = {X 454.1396, Y 97.0659, Z -7.1667, A 0.000, B 0.000, C 0.000 }
gfCNCPoint5[21197] = {X 454.2295, Y 96.1891, Z -7.1667, A 0.000, B 0.000, C 0.000 }
gfCNCPoint5[21198] = {X 454.4955, Y 95.3488, Z -7.1667, A 0.000, B 0.000, C 0.000 }
gfCNCPoint5[21199] = {X 454.9265, Y 94.5800, Z -7.1667, A 0.000, B 0.000, C 0.000 }
gfCNCPoint5[21200] = {X 455.5046, Y 93.9147, Z -7.1667, A 0.000, B 0.000, C 0.000 }
gfCNCPoint5[21201] = {X 456.2057, Y 93.3805, Z -7.1667, A 0.000, B 0.000, C 0.000 }
gfCNCPoint5[21202] = {X 457.0006, Y 92.9998, Z -7.1667, A 0.000, B 0.000, C 0.000 }
gfCNCPoint5[21203] = {X 457.8563, Y 92.7883, Z -7.1667, A 0.000, B 0.000, C 0.000 }
gfCNCPoint5[21204] = {X 457.8563, Y 85.5950, Z -7.1667, A 0.000, B 0.000, C 0.000 }
gfCNCPoint5[21205] = {X 444.8602, Y 80.5005, Z -7.1667, A 0.000, B 0.000, C 0.000 }
gfCNCPoint5[21206] = {X 420.0242, Y 96.5885, Z -7.1667, A 0.000, B 0.000, C 0.000 }
gfCNCPoint5[21207] = {X 420.0267, Y 97.0651, Z -7.1667, A 0.000, B 0.000, C 0.000 }
gfCNCPoint5[21208] = {X 420.0267, Y 98.0000, Z -7.1667, A 0.000, B 0.000, C 0.000 }
gfCNCPoint5[21209] = {X 419.9184, Y 98.9613, Z -7.1667, A 0.000, B 0.000, C 0.000 }
gfCNCPoint5[21210] = {X 419.5989, Y 99.8744, Z -7.1667, A 0.000, B 0.000, C 0.000 }
gfCNCPoint5[21211] = {X 419.0842, Y 100.6935, Z -7.1667, A 0.000, B 0.000, C 0.000 }
gfCNCPoint5[21212] = {X 418.4002, Y 101.3775, Z -7.1667, A 0.000, B 0.000, C 0.000 }
gfCNCPoint5[21213] = {X 417.5811, Y 101.8922, Z -7.1667, A 0.000, B 0.000, C 0.000 }
gfCNCPoint5[21214] = {X 416.6680, Y 102.2117, Z -7.1667, A 0.000, B 0.000, C 0.000 }
gfCNCPoint5[21215] = {X 415.7067, Y 102.3200, Z -7.1667, A 0.000, B 0.000, C 0.000 }
gfCNCPoint5[21216] = {X 396.4059, Y 102.3200, Z -7.1667, A 0.000, B 0.000, C 0.000 }
gfCNCPoint5[21217] = {X 395.4447, Y 102.2117, Z -7.1667, A 0.000, B 0.000, C 0.000 }
gfCNCPoint5[21218] = {X 394.5316, Y 101.8922, Z -7.1667, A 0.000, B 0.000, C 0.000 }
gfCNCPoint5[21219] = {X 393.7125, Y 101.3775, Z -7.1667, A 0.000, B 0.000, C 0.000 }
gfCNCPoint5[21220] = {X 393.0284, Y 100.6935, Z -7.1667, A 0.000, B 0.000, C 0.000 }
gfCNCPoint5[21221] = {X 392.5138, Y 99.8744, Z -7.1667, A 0.000, B 0.000, C 0.000 }
gfCNCPoint5[21222] = {X 392.1943, Y 98.9613, Z -7.1667, A 0.000, B 0.000, C 0.000 }
gfCNCPoint5[21223] = {X 392.0859, Y 98.0000, Z -7.1667, A 0.000, B 0.000, C 0.000 }
gfCNCPoint5[21224] = {X 392.0859, Y 97.0659, Z -7.1667, A 0.000, B 0.000, C 0.000 }
gfCNCPoint5[21225] = {X 392.1940, Y 96.1060, Z -7.1667, A 0.000, B 0.000, C 0.000 }
gfCNCPoint5[21226] = {X 392.5126, Y 95.1940, Z -7.1667, A 0.000, B 0.000, C 0.000 }
gfCNCPoint5[21227] = {X 393.0259, Y 94.3757, Z -7.1667, A 0.000, B 0.000, C 0.000 }
gfCNCPoint5[21228] = {X 393.7082, Y 93.6918, Z -7.1667, A 0.000, B 0.000, C 0.000 }
gfCNCPoint5[21229] = {X 394.5254, Y 93.1767, Z -7.1667, A 0.000, B 0.000, C 0.000 }
gfCNCPoint5[21230] = {X 395.4367, Y 92.8561, Z -7.1667, A 0.000, B 0.000, C 0.000 }
gfCNCPoint5[21231] = {X 396.3964, Y 92.7459, Z -7.1667, A 0.000, B 0.000, C 0.000 }
gfCNCPoint5[21232] = {X 397.3466, Y 92.7030, Z -7.1667, A 0.000, B 0.000, C 0.000 }
gfCNCPoint5[21233] = {X 398.2935, Y 92.6133, Z -7.1667, A 0.000, B 0.000, C 0.000 }
gfCNCPoint5[21234] = {X 398.9444, Y 92.4554, Z -7.1667, A 0.000, B 0.000, C 0.000 }
gfCNCPoint5[21235] = {X 399.5438, Y 92.1566, Z -7.1667, A 0.000, B 0.000, C 0.000 }
gfCNCPoint5[21236] = {X 413.7986, Y 83.0281, Z -7.1667, A 0.000, B 0.000, C 0.000 }
gfCNCPoint5[21237] = {X 411.6415, Y 79.6596, Z -7.1667, A 0.000, B 0.000, C 0.000 }
gfCNCPoint5[21238] = {X 413.8418, Y 83.0955, Z -7.1667, A 0.000, B 0.000, C 0.000 }
gfCNCPoint5[21239] = {X 428.2287, Y 73.8824, Z -7.1667, A 0.000, B 0.000, C 0.000 }
gfCNCPoint5[21240] = {X 403.7848, Y 64.2924, Z -7.1667, A 0.000, B 0.000, C 0.000 }
gfCNCPoint5[21241] = {X 402.0799, Y 63.7281, Z -7.1667, A 0.000, B 0.000, C 0.000 }
gfCNCPoint5[21242] = {X 400.3235, Y 63.3538, Z -7.1667, A 0.000, B 0.000, C 0.000 }
gfCNCPoint5[21243] = {X 398.5367, Y 63.1740, Z -7.1667, A 0.000, B 0.000, C 0.000 }
gfCNCPoint5[21244] = {X 397.6016, Y 63.0649, Z -7.1667, A 0.000, B 0.000, C 0.000 }
gfCNCPoint5[21245] = {X 396.7136, Y 62.7520, Z -7.1667, A 0.000, B 0.000, C 0.000 }
gfCNCPoint5[21246] = {X 395.9165, Y 62.2509, Z -7.1667, A 0.000, B 0.000, C 0.000 }
gfCNCPoint5[21247] = {X 395.2496, Y 61.5863, Z -7.1667, A 0.000, B 0.000, C 0.000 }
gfCNCPoint5[21248] = {X 394.7459, Y 60.7908, Z -7.1667, A 0.000, B 0.000, C 0.000 }
gfCNCPoint5[21249] = {X 394.4301, Y 59.9039, Z -7.1667, A 0.000, B 0.000, C 0.000 }
gfCNCPoint5[21250] = {X 394.3179, Y 58.9691, Z -7.1667, A 0.000, B 0.000, C 0.000 }
gfCNCPoint5[21251] = {X 394.3177, Y 58.0000, Z -7.1667, A 0.000, B 0.000, C 0.000 }
gfCNCPoint5[21252] = {X 394.4240, Y 57.0565, Z -7.1667, A 0.000, B 0.000, C 0.000 }
gfCNCPoint5[21253] = {X 394.7376, Y 56.1603, Z -7.1667, A 0.000, B 0.000, C 0.000 }
gfCNCPoint5[21254] = {X 395.2428, Y 55.3564, Z -7.1667, A 0.000, B 0.000, C 0.000 }
gfCNCPoint5[21255] = {X 395.9141, Y 54.6850, Z -7.1667, A 0.000, B 0.000, C 0.000 }
gfCNCPoint5[21256] = {X 396.7181, Y 54.1799, Z -7.1667, A 0.000, B 0.000, C 0.000 }
gfCNCPoint5[21257] = {X 397.6142, Y 53.8663, Z -7.1667, A 0.000, B 0.000, C 0.000 }
gfCNCPoint5[21258] = {X 398.5577, Y 53.7600, Z -7.1667, A 0.000, B 0.000, C 0.000 }
gfCNCPoint5[21259] = {X 419.4886, Y 53.7600, Z -7.1667, A 0.000, B 0.000, C 0.000 }
gfCNCPoint5[21260] = {X 420.4321, Y 53.8663, Z -7.1667, A 0.000, B 0.000, C 0.000 }
gfCNCPoint5[21261] = {X 421.3283, Y 54.1799, Z -7.1667, A 0.000, B 0.000, C 0.000 }
gfCNCPoint5[21262] = {X 422.1322, Y 54.6850, Z -7.1667, A 0.000, B 0.000, C 0.000 }
gfCNCPoint5[21263] = {X 422.8036, Y 55.3564, Z -7.1667, A 0.000, B 0.000, C 0.000 }
gfCNCPoint5[21264] = {X 423.3087, Y 56.1603, Z -7.1667, A 0.000, B 0.000, C 0.000 }
gfCNCPoint5[21265] = {X 423.6223, Y 57.0565, Z -7.1667, A 0.000, B 0.000, C 0.000 }
gfCNCPoint5[21266] = {X 423.7286, Y 58.0000, Z -7.1667, A 0.000, B 0.000, C 0.000 }
gfCNCPoint5[21267] = {X 423.7286, Y 58.2862, Z -7.1667, A 0.000, B 0.000, C 0.000 }
gfCNCPoint5[21268] = {X 429.5823, Y 60.5668, Z -7.1667, A 0.000, B 0.000, C 0.000 }
gfCNCPoint5[21269] = {X 457.9380, Y 71.8176, Z -7.1667, A 0.000, B 0.000, C 0.000 }
gfCNCPoint5[21270] = {X 457.9402, Y 63.1421, Z -7.1667, A 0.000, B 0.000, C 0.000 }
gfCNCPoint5[21271] = {X 457.0918, Y 62.9474, Z -7.1667, A 0.000, B 0.000, C 0.000 }
gfCNCPoint5[21272] = {X 456.3010, Y 62.5834, Z -7.1667, A 0.000, B 0.000, C 0.000 }
gfCNCPoint5[21273] = {X 455.6012, Y 62.0657, Z -7.1667, A 0.000, B 0.000, C 0.000 }
gfCNCPoint5[21274] = {X 455.0218, Y 61.4159, Z -7.1667, A 0.000, B 0.000, C 0.000 }
gfCNCPoint5[21275] = {X 454.5874, Y 60.6615, Z -7.1667, A 0.000, B 0.000, C 0.000 }
gfCNCPoint5[21276] = {X 454.3163, Y 59.8342, Z -7.1667, A 0.000, B 0.000, C 0.000 }
gfCNCPoint5[21277] = {X 454.2197, Y 58.9691, Z -7.1667, A 0.000, B 0.000, C 0.000 }
gfCNCPoint5[21278] = {X 454.2196, Y 58.0000, Z -7.1667, A 0.000, B 0.000, C 0.000 }
gfCNCPoint5[21279] = {X 454.3259, Y 57.0565, Z -7.1667, A 0.000, B 0.000, C 0.000 }
gfCNCPoint5[21280] = {X 454.6395, Y 56.1603, Z -7.1667, A 0.000, B 0.000, C 0.000 }
gfCNCPoint5[21281] = {X 455.1446, Y 55.3564, Z -7.1667, A 0.000, B 0.000, C 0.000 }
gfCNCPoint5[21282] = {X 455.8160, Y 54.6850, Z -7.1667, A 0.000, B 0.000, C 0.000 }
gfCNCPoint5[21283] = {X 456.6199, Y 54.1799, Z -7.1667, A 0.000, B 0.000, C 0.000 }
gfCNCPoint5[21284] = {X 457.5161, Y 53.8663, Z -7.1667, A 0.000, B 0.000, C 0.000 }
gfCNCPoint5[21285] = {X 458.4596, Y 53.7600, Z -7.1667, A 0.000, B 0.000, C 0.000 }
gfCNCPoint5[21286] = {X 475.0000, Y 53.7600, Z -7.1667, A 0.000, B 0.000, C 0.000 }
gfCNCPoint5[21287] = {X 475.9435, Y 53.8663, Z -7.1667, A 0.000, B 0.000, C 0.000 }
gfCNCPoint5[21288] = {X 476.8397, Y 54.1799, Z -7.1667, A 0.000, B 0.000, C 0.000 }
gfCNCPoint5[21289] = {X 477.6436, Y 54.6850, Z -7.1667, A 0.000, B 0.000, C 0.000 }
gfCNCPoint5[21290] = {X 478.3150, Y 55.3564, Z -7.1667, A 0.000, B 0.000, C 0.000 }
gfCNCPoint5[21291] = {X 478.8201, Y 56.1603, Z -7.1667, A 0.000, B 0.000, C 0.000 }
gfCNCPoint5[21292] = {X 479.1337, Y 57.0565, Z -7.1667, A 0.000, B 0.000, C 0.000 }
gfCNCPoint5[21293] = {X 479.2400, Y 58.0000, Z -7.1667, A 0.000, B 0.000, C 0.000 }
gfCNCPoint5[21294] = {X 479.2400, Y 58.9342, Z -7.1667, A 0.000, B 0.000, C 0.000 }
gfCNCPoint5[21295] = {X 479.1496, Y 59.8048, Z -7.1667, A 0.000, B 0.000, C 0.000 }
gfCNCPoint5[21296] = {X 478.8824, Y 60.6383, Z -7.1667, A 0.000, B 0.000, C 0.000 }
gfCNCPoint5[21297] = {X 478.4498, Y 61.3991, Z -7.1667, A 0.000, B 0.000, C 0.000 }
gfCNCPoint5[21298] = {X 477.8702, Y 62.0549, Z -7.1667, A 0.000, B 0.000, C 0.000 }
gfCNCPoint5[21299] = {X 477.1682, Y 62.5778, Z -7.1667, A 0.000, B 0.000, C 0.000 }
gfCNCPoint5[21300] = {X 476.3739, Y 62.9453, Z -7.1667, A 0.000, B 0.000, C 0.000 }
gfCNCPoint5[21301] = {X 475.5210, Y 63.1419, Z -7.1667, A 0.000, B 0.000, C 0.000 }
gfCNCPoint5[21302] = {X 475.5214, Y 92.8318, Z -7.1667, A 0.000, B 0.000, C 0.000 }
gfCNCPoint5[21303] = {X 475.9412, Y 92.9338, Z -7.1667, A 0.000, B 0.000, C 0.000 }
gfCNCPoint5[21304] = {X 476.3547, Y 93.0589, Z -7.1667, A 0.000, B 0.000, C 0.000 }
gfCNCPoint5[21305] = {X 477.1532, Y 93.4209, Z -7.1667, A 0.000, B 0.000, C 0.000 }
gfCNCPoint5[21306] = {X 477.8596, Y 93.9402, Z -7.1667, A 0.000, B 0.000, C 0.000 }
gfCNCPoint5[21307] = {X 478.4435, Y 94.5942, Z -7.1667, A 0.000, B 0.000, C 0.000 }
gfCNCPoint5[21308] = {X 478.8795, Y 95.3549, Z -7.1667, A 0.000, B 0.000, C 0.000 }
gfCNCPoint5[21309] = {X 479.1489, Y 96.1892, Z -7.1667, A 0.000, B 0.000, C 0.000 }
gfCNCPoint5[21310] = {X 479.2400, Y 97.0611, Z -7.1667, A 0.000, B 0.000, C 0.000 }
gfCNCPoint5[21311] = {X 479.2400, Y 98.0000, Z -7.1667, A 0.000, B 0.000, C 0.000 }
gfCNCPoint5[21312] = {X 479.1337, Y 98.9435, Z -7.1667, A 0.000, B 0.000, C 0.000 }
gfCNCPoint5[21313] = {X 478.8201, Y 99.8397, Z -7.1667, A 0.000, B 0.000, C 0.000 }
gfCNCPoint5[21314] = {X 478.3150, Y 100.6436, Z -7.1667, A 0.000, B 0.000, C 0.000 }
gfCNCPoint5[21315] = {X 477.6436, Y 101.3150, Z -7.1667, A 0.000, B 0.000, C 0.000 }
gfCNCPoint5[21316] = {X 476.8397, Y 101.8201, Z -7.1667, A 0.000, B 0.000, C 0.000 }
gfCNCPoint5[21317] = {X 475.9435, Y 102.1337, Z -7.1667, A 0.000, B 0.000, C 0.000 }
gfCNCPoint5[21318] = {X 475.0000, Y 102.2400, Z -7.1667, A 0.000, B 0.000, C 0.000 }
gfCNCPoint5[21319] = {X 458.4596, Y 102.2400, Z -7.1667, A 0.000, B 0.000, C 0.000 }
gfCNCPoint5[21320] = {X 457.5161, Y 102.1337, Z -7.1667, A 0.000, B 0.000, C 0.000 }
gfCNCPoint5[21321] = {X 456.6199, Y 101.8201, Z -7.1667, A 0.000, B 0.000, C 0.000 }
gfCNCPoint5[21322] = {X 455.8160, Y 101.3150, Z -7.1667, A 0.000, B 0.000, C 0.000 }
gfCNCPoint5[21323] = {X 455.1446, Y 100.6436, Z -7.1667, A 0.000, B 0.000, C 0.000 }
gfCNCPoint5[21324] = {X 454.6395, Y 99.8397, Z -7.1667, A 0.000, B 0.000, C 0.000 }
gfCNCPoint5[21325] = {X 454.3259, Y 98.9435, Z -7.1667, A 0.000, B 0.000, C 0.000 }
gfCNCPoint5[21326] = {X 454.2196, Y 98.0000, Z -7.1667, A 0.000, B 0.000, C 0.000 }
gfCNCPoint5[21327] = {X 454.2196, Y 97.0659, Z -7.1667, A 0.000, B 0.000, C 0.000 }
gfCNCPoint5[21328] = {X 454.3099, Y 96.1957, Z -7.1667, A 0.000, B 0.000, C 0.000 }
gfCNCPoint5[21329] = {X 454.5769, Y 95.3624, Z -7.1667, A 0.000, B 0.000, C 0.000 }
gfCNCPoint5[21330] = {X 455.0092, Y 94.6018, Z -7.1667, A 0.000, B 0.000, C 0.000 }
gfCNCPoint5[21331] = {X 455.5884, Y 93.9460, Z -7.1667, A 0.000, B 0.000, C 0.000 }
gfCNCPoint5[21332] = {X 456.2899, Y 93.4231, Z -7.1667, A 0.000, B 0.000, C 0.000 }
gfCNCPoint5[21333] = {X 457.0838, Y 93.0553, Z -7.1667, A 0.000, B 0.000, C 0.000 }
gfCNCPoint5[21334] = {X 457.9363, Y 92.8584, Z -7.1667, A 0.000, B 0.000, C 0.000 }
gfCNCPoint5[21335] = {X 457.9363, Y 85.5404, Z -7.1667, A 0.000, B 0.000, C 0.000 }
gfCNCPoint5[21336] = {X 444.8511, Y 80.4110, Z -7.1667, A 0.000, B 0.000, C 0.000 }
gfCNCPoint5[21337] = {X 419.9440, Y 96.5451, Z -7.1667, A 0.000, B 0.000, C 0.000 }
gfCNCPoint5[21338] = {X 419.9467, Y 97.0653, Z -7.1667, A 0.000, B 0.000, C 0.000 }
gfCNCPoint5[21339] = {X 419.9467, Y 98.0000, Z -7.1667, A 0.000, B 0.000, C 0.000 }
gfCNCPoint5[21340] = {X 419.8404, Y 98.9435, Z -7.1667, A 0.000, B 0.000, C 0.000 }
gfCNCPoint5[21341] = {X 419.5268, Y 99.8397, Z -7.1667, A 0.000, B 0.000, C 0.000 }
gfCNCPoint5[21342] = {X 419.0217, Y 100.6436, Z -7.1667, A 0.000, B 0.000, C 0.000 }
gfCNCPoint5[21343] = {X 418.3503, Y 101.3150, Z -7.1667, A 0.000, B 0.000, C 0.000 }
gfCNCPoint5[21344] = {X 417.5464, Y 101.8201, Z -7.1667, A 0.000, B 0.000, C 0.000 }
gfCNCPoint5[21345] = {X 416.6502, Y 102.1337, Z -7.1667, A 0.000, B 0.000, C 0.000 }
gfCNCPoint5[21346] = {X 415.7067, Y 102.2400, Z -7.1667, A 0.000, B 0.000, C 0.000 }
gfCNCPoint5[21347] = {X 396.4059, Y 102.2400, Z -7.1667, A 0.000, B 0.000, C 0.000 }
gfCNCPoint5[21348] = {X 395.4625, Y 102.1337, Z -7.1667, A 0.000, B 0.000, C 0.000 }
gfCNCPoint5[21349] = {X 394.5663, Y 101.8201, Z -7.1667, A 0.000, B 0.000, C 0.000 }
gfCNCPoint5[21350] = {X 393.7624, Y 101.3150, Z -7.1667, A 0.000, B 0.000, C 0.000 }
gfCNCPoint5[21351] = {X 393.0910, Y 100.6436, Z -7.1667, A 0.000, B 0.000, C 0.000 }
gfCNCPoint5[21352] = {X 392.5858, Y 99.8397, Z -7.1667, A 0.000, B 0.000, C 0.000 }
gfCNCPoint5[21353] = {X 392.2723, Y 98.9435, Z -7.1667, A 0.000, B 0.000, C 0.000 }
gfCNCPoint5[21354] = {X 392.1659, Y 98.0000, Z -7.1667, A 0.000, B 0.000, C 0.000 }
gfCNCPoint5[21355] = {X 392.1659, Y 97.0659, Z -7.1667, A 0.000, B 0.000, C 0.000 }
gfCNCPoint5[21356] = {X 392.2720, Y 96.1236, Z -7.1667, A 0.000, B 0.000, C 0.000 }
gfCNCPoint5[21357] = {X 392.5848, Y 95.2285, Z -7.1667, A 0.000, B 0.000, C 0.000 }
gfCNCPoint5[21358] = {X 393.0887, Y 94.4252, Z -7.1667, A 0.000, B 0.000, C 0.000 }
gfCNCPoint5[21359] = {X 393.7585, Y 93.7540, Z -7.1667, A 0.000, B 0.000, C 0.000 }
gfCNCPoint5[21360] = {X 394.5607, Y 93.2485, Z -7.1667, A 0.000, B 0.000, C 0.000 }
gfCNCPoint5[21361] = {X 395.4552, Y 92.9339, Z -7.1667, A 0.000, B 0.000, C 0.000 }
gfCNCPoint5[21362] = {X 396.3973, Y 92.8259, Z -7.1667, A 0.000, B 0.000, C 0.000 }
gfCNCPoint5[21363] = {X 397.3520, Y 92.7829, Z -7.1667, A 0.000, B 0.000, C 0.000 }
gfCNCPoint5[21364] = {X 398.3033, Y 92.6927, Z -7.1667, A 0.000, B 0.000, C 0.000 }
gfCNCPoint5[21365] = {X 398.9717, Y 92.5306, Z -7.1667, A 0.000, B 0.000, C 0.000 }
gfCNCPoint5[21366] = {X 399.5872, Y 92.2237, Z -7.1667, A 0.000, B 0.000, C 0.000 }
gfCNCPoint5[21367] = {X 413.8418, Y 83.0955, Z -7.1667, A 0.000, B 0.000, C 0.000 }
gfCNCPoint5[21368] = {X 411.6847, Y 79.7270, Z -7.1667, A 0.000, B 0.000, C 0.000 }
gfCNCPoint5[21369] = {X 413.8849, Y 83.1628, Z -7.1667, A 0.000, B 0.000, C 0.000 }
gfCNCPoint5[21370] = {X 428.4039, Y 73.8652, Z -7.1667, A 0.000, B 0.000, C 0.000 }
gfCNCPoint5[21371] = {X 403.8141, Y 64.2180, Z -7.1667, A 0.000, B 0.000, C 0.000 }
gfCNCPoint5[21372] = {X 402.1004, Y 63.6508, Z -7.1667, A 0.000, B 0.000, C 0.000 }
gfCNCPoint5[21373] = {X 400.3348, Y 63.2746, Z -7.1667, A 0.000, B 0.000, C 0.000 }
gfCNCPoint5[21374] = {X 398.5388, Y 63.0940, Z -7.1667, A 0.000, B 0.000, C 0.000 }
gfCNCPoint5[21375] = {X 397.6210, Y 62.9872, Z -7.1667, A 0.000, B 0.000, C 0.000 }
gfCNCPoint5[21376] = {X 396.7494, Y 62.6805, Z -7.1667, A 0.000, B 0.000, C 0.000 }
gfCNCPoint5[21377] = {X 395.9670, Y 62.1889, Z -7.1667, A 0.000, B 0.000, C 0.000 }
gfCNCPoint5[21378] = {X 395.3125, Y 61.5368, Z -7.1667, A 0.000, B 0.000, C 0.000 }
gfCNCPoint5[21379] = {X 394.8180, Y 60.7562, Z -7.1667, A 0.000, B 0.000, C 0.000 }
gfCNCPoint5[21380] = {X 394.5081, Y 59.8858, Z -7.1667, A 0.000, B 0.000, C 0.000 }
gfCNCPoint5[21381] = {X 394.3979, Y 58.9684, Z -7.1667, A 0.000, B 0.000, C 0.000 }
gfCNCPoint5[21382] = {X 394.3977, Y 58.0000, Z -7.1667, A 0.000, B 0.000, C 0.000 }
gfCNCPoint5[21383] = {X 394.5020, Y 57.0743, Z -7.1667, A 0.000, B 0.000, C 0.000 }
gfCNCPoint5[21384] = {X 394.8097, Y 56.1950, Z -7.1667, A 0.000, B 0.000, C 0.000 }
gfCNCPoint5[21385] = {X 395.3053, Y 55.4063, Z -7.1667, A 0.000, B 0.000, C 0.000 }
gfCNCPoint5[21386] = {X 395.9640, Y 54.7476, Z -7.1667, A 0.000, B 0.000, C 0.000 }
gfCNCPoint5[21387] = {X 396.7528, Y 54.2520, Z -7.1667, A 0.000, B 0.000, C 0.000 }
gfCNCPoint5[21388] = {X 397.6320, Y 53.9443, Z -7.1667, A 0.000, B 0.000, C 0.000 }
gfCNCPoint5[21389] = {X 398.5577, Y 53.8400, Z -7.1667, A 0.000, B 0.000, C 0.000 }
gfCNCPoint5[21390] = {X 419.4886, Y 53.8400, Z -7.1667, A 0.000, B 0.000, C 0.000 }
gfCNCPoint5[21391] = {X 420.4143, Y 53.9443, Z -7.1667, A 0.000, B 0.000, C 0.000 }
gfCNCPoint5[21392] = {X 421.2936, Y 54.2520, Z -7.1667, A 0.000, B 0.000, C 0.000 }
gfCNCPoint5[21393] = {X 422.0823, Y 54.7476, Z -7.1667, A 0.000, B 0.000, C 0.000 }
gfCNCPoint5[21394] = {X 422.7410, Y 55.4063, Z -7.1667, A 0.000, B 0.000, C 0.000 }
gfCNCPoint5[21395] = {X 423.2366, Y 56.1950, Z -7.1667, A 0.000, B 0.000, C 0.000 }
gfCNCPoint5[21396] = {X 423.5443, Y 57.0743, Z -7.1667, A 0.000, B 0.000, C 0.000 }
gfCNCPoint5[21397] = {X 423.6486, Y 58.0000, Z -7.1667, A 0.000, B 0.000, C 0.000 }
gfCNCPoint5[21398] = {X 423.6486, Y 58.3409, Z -7.1667, A 0.000, B 0.000, C 0.000 }
gfCNCPoint5[21399] = {X 429.5530, Y 60.6413, Z -7.1667, A 0.000, B 0.000, C 0.000 }
gfCNCPoint5[21400] = {X 458.0180, Y 71.9354, Z -7.1667, A 0.000, B 0.000, C 0.000 }
gfCNCPoint5[21401] = {X 458.0203, Y 63.0708, Z -7.1667, A 0.000, B 0.000, C 0.000 }
gfCNCPoint5[21402] = {X 457.9177, Y 63.0586, Z -7.1667, A 0.000, B 0.000, C 0.000 }
gfCNCPoint5[21403] = {X 457.8155, Y 63.0439, Z -7.1667, A 0.000, B 0.000, C 0.000 }
gfCNCPoint5[21404] = {X 456.8781, Y 62.7817, Z -7.1667, A 0.000, B 0.000, C 0.000 }
gfCNCPoint5[21405] = {X 456.0273, Y 62.3089, Z -7.1667, A 0.000, B 0.000, C 0.000 }
gfCNCPoint5[21406] = {X 455.3097, Y 61.6513, Z -7.1667, A 0.000, B 0.000, C 0.000 }
gfCNCPoint5[21407] = {X 454.7645, Y 60.8450, Z -7.1667, A 0.000, B 0.000, C 0.000 }
gfCNCPoint5[21408] = {X 454.4216, Y 59.9341, Z -7.1667, A 0.000, B 0.000, C 0.000 }
gfCNCPoint5[21409] = {X 454.2997, Y 58.9684, Z -7.1667, A 0.000, B 0.000, C 0.000 }
gfCNCPoint5[21410] = {X 454.2996, Y 58.0000, Z -7.1667, A 0.000, B 0.000, C 0.000 }
gfCNCPoint5[21411] = {X 454.4039, Y 57.0743, Z -7.1667, A 0.000, B 0.000, C 0.000 }
gfCNCPoint5[21412] = {X 454.7116, Y 56.1950, Z -7.1667, A 0.000, B 0.000, C 0.000 }
gfCNCPoint5[21413] = {X 455.2072, Y 55.4063, Z -7.1667, A 0.000, B 0.000, C 0.000 }
gfCNCPoint5[21414] = {X 455.8659, Y 54.7476, Z -7.1667, A 0.000, B 0.000, C 0.000 }
gfCNCPoint5[21415] = {X 456.6546, Y 54.2520, Z -7.1667, A 0.000, B 0.000, C 0.000 }
gfCNCPoint5[21416] = {X 457.5339, Y 53.9443, Z -7.1667, A 0.000, B 0.000, C 0.000 }
gfCNCPoint5[21417] = {X 458.4596, Y 53.8400, Z -7.1667, A 0.000, B 0.000, C 0.000 }
gfCNCPoint5[21418] = {X 475.0000, Y 53.8400, Z -7.1667, A 0.000, B 0.000, C 0.000 }
gfCNCPoint5[21419] = {X 475.9257, Y 53.9443, Z -7.1667, A 0.000, B 0.000, C 0.000 }
gfCNCPoint5[21420] = {X 476.8050, Y 54.2520, Z -7.1667, A 0.000, B 0.000, C 0.000 }
gfCNCPoint5[21421] = {X 477.5937, Y 54.7476, Z -7.1667, A 0.000, B 0.000, C 0.000 }
gfCNCPoint5[21422] = {X 478.2524, Y 55.4063, Z -7.1667, A 0.000, B 0.000, C 0.000 }
gfCNCPoint5[21423] = {X 478.7480, Y 56.1950, Z -7.1667, A 0.000, B 0.000, C 0.000 }
gfCNCPoint5[21424] = {X 479.0557, Y 57.0743, Z -7.1667, A 0.000, B 0.000, C 0.000 }
gfCNCPoint5[21425] = {X 479.1600, Y 58.0000, Z -7.1667, A 0.000, B 0.000, C 0.000 }
gfCNCPoint5[21426] = {X 479.1600, Y 58.9342, Z -7.1667, A 0.000, B 0.000, C 0.000 }
gfCNCPoint5[21427] = {X 479.0448, Y 59.9065, Z -7.1667, A 0.000, B 0.000, C 0.000 }
gfCNCPoint5[21428] = {X 478.7055, Y 60.8248, Z -7.1667, A 0.000, B 0.000, C 0.000 }
gfCNCPoint5[21429] = {X 478.1610, Y 61.6385, Z -7.1667, A 0.000, B 0.000, C 0.000 }
gfCNCPoint5[21430] = {X 477.4414, Y 62.3024, Z -7.1667, A 0.000, B 0.000, C 0.000 }
gfCNCPoint5[21431] = {X 476.5865, Y 62.7796, Z -7.1667, A 0.000, B 0.000, C 0.000 }
gfCNCPoint5[21432] = {X 475.6438, Y 63.0439, Z -7.1667, A 0.000, B 0.000, C 0.000 }
gfCNCPoint5[21433] = {X 475.5426, Y 63.0585, Z -7.1667, A 0.000, B 0.000, C 0.000 }
gfCNCPoint5[21434] = {X 475.4410, Y 63.0706, Z -7.1667, A 0.000, B 0.000, C 0.000 }
gfCNCPoint5[21435] = {X 475.4414, Y 92.8968, Z -7.1667, A 0.000, B 0.000, C 0.000 }
gfCNCPoint5[21436] = {X 475.8890, Y 93.0026, Z -7.1667, A 0.000, B 0.000, C 0.000 }
gfCNCPoint5[21437] = {X 476.3294, Y 93.1348, Z -7.1667, A 0.000, B 0.000, C 0.000 }
gfCNCPoint5[21438] = {X 477.1128, Y 93.4900, Z -7.1667, A 0.000, B 0.000, C 0.000 }
gfCNCPoint5[21439] = {X 477.8058, Y 93.9994, Z -7.1667, A 0.000, B 0.000, C 0.000 }
gfCNCPoint5[21440] = {X 478.3786, Y 94.6410, Z -7.1667, A 0.000, B 0.000, C 0.000 }
gfCNCPoint5[21441] = {X 478.8063, Y 95.3872, Z -7.1667, A 0.000, B 0.000, C 0.000 }
gfCNCPoint5[21442] = {X 479.0706, Y 96.2057, Z -7.1667, A 0.000, B 0.000, C 0.000 }
gfCNCPoint5[21443] = {X 479.1600, Y 97.0611, Z -7.1667, A 0.000, B 0.000, C 0.000 }
gfCNCPoint5[21444] = {X 479.1600, Y 98.0000, Z -7.1667, A 0.000, B 0.000, C 0.000 }
gfCNCPoint5[21445] = {X 479.0557, Y 98.9257, Z -7.1667, A 0.000, B 0.000, C 0.000 }
gfCNCPoint5[21446] = {X 478.7480, Y 99.8050, Z -7.1667, A 0.000, B 0.000, C 0.000 }
gfCNCPoint5[21447] = {X 478.2524, Y 100.5937, Z -7.1667, A 0.000, B 0.000, C 0.000 }
gfCNCPoint5[21448] = {X 477.5937, Y 101.2524, Z -7.1667, A 0.000, B 0.000, C 0.000 }
gfCNCPoint5[21449] = {X 476.8050, Y 101.7480, Z -7.1667, A 0.000, B 0.000, C 0.000 }
gfCNCPoint5[21450] = {X 475.9257, Y 102.0557, Z -7.1667, A 0.000, B 0.000, C 0.000 }
gfCNCPoint5[21451] = {X 475.0000, Y 102.1600, Z -7.1667, A 0.000, B 0.000, C 0.000 }
gfCNCPoint5[21452] = {X 458.4596, Y 102.1600, Z -7.1667, A 0.000, B 0.000, C 0.000 }
gfCNCPoint5[21453] = {X 457.5339, Y 102.0557, Z -7.1667, A 0.000, B 0.000, C 0.000 }
gfCNCPoint5[21454] = {X 456.6546, Y 101.7480, Z -7.1667, A 0.000, B 0.000, C 0.000 }
gfCNCPoint5[21455] = {X 455.8659, Y 101.2524, Z -7.1667, A 0.000, B 0.000, C 0.000 }
gfCNCPoint5[21456] = {X 455.2072, Y 100.5937, Z -7.1667, A 0.000, B 0.000, C 0.000 }
gfCNCPoint5[21457] = {X 454.7116, Y 99.8050, Z -7.1667, A 0.000, B 0.000, C 0.000 }
gfCNCPoint5[21458] = {X 454.4039, Y 98.9257, Z -7.1667, A 0.000, B 0.000, C 0.000 }
gfCNCPoint5[21459] = {X 454.2996, Y 98.0000, Z -7.1667, A 0.000, B 0.000, C 0.000 }
gfCNCPoint5[21460] = {X 454.2996, Y 97.0659, Z -7.1667, A 0.000, B 0.000, C 0.000 }
gfCNCPoint5[21461] = {X 454.3903, Y 96.2022, Z -7.1667, A 0.000, B 0.000, C 0.000 }
gfCNCPoint5[21462] = {X 454.6583, Y 95.3761, Z -7.1667, A 0.000, B 0.000, C 0.000 }
gfCNCPoint5[21463] = {X 455.0920, Y 94.6237, Z -7.1667, A 0.000, B 0.000, C 0.000 }
gfCNCPoint5[21464] = {X 455.6724, Y 93.9777, Z -7.1667, A 0.000, B 0.000, C 0.000 }
gfCNCPoint5[21465] = {X 456.3743, Y 93.4663, Z -7.1667, A 0.000, B 0.000, C 0.000 }
gfCNCPoint5[21466] = {X 457.1672, Y 93.1118, Z -7.1667, A 0.000, B 0.000, C 0.000 }
gfCNCPoint5[21467] = {X 458.0163, Y 92.9296, Z -7.1667, A 0.000, B 0.000, C 0.000 }
gfCNCPoint5[21468] = {X 458.0163, Y 85.4858, Z -7.1667, A 0.000, B 0.000, C 0.000 }
gfCNCPoint5[21469] = {X 444.8421, Y 80.3215, Z -7.1667, A 0.000, B 0.000, C 0.000 }
gfCNCPoint5[21470] = {X 419.8637, Y 96.5018, Z -7.1667, A 0.000, B 0.000, C 0.000 }
gfCNCPoint5[21471] = {X 419.8667, Y 97.0655, Z -7.1667, A 0.000, B 0.000, C 0.000 }
gfCNCPoint5[21472] = {X 419.8667, Y 98.0000, Z -7.1667, A 0.000, B 0.000, C 0.000 }
gfCNCPoint5[21473] = {X 419.7624, Y 98.9257, Z -7.1667, A 0.000, B 0.000, C 0.000 }
gfCNCPoint5[21474] = {X 419.4547, Y 99.8050, Z -7.1667, A 0.000, B 0.000, C 0.000 }
gfCNCPoint5[21475] = {X 418.9591, Y 100.5937, Z -7.1667, A 0.000, B 0.000, C 0.000 }
gfCNCPoint5[21476] = {X 418.3004, Y 101.2524, Z -7.1667, A 0.000, B 0.000, C 0.000 }
gfCNCPoint5[21477] = {X 417.5117, Y 101.7480, Z -7.1667, A 0.000, B 0.000, C 0.000 }
gfCNCPoint5[21478] = {X 416.6324, Y 102.0557, Z -7.1667, A 0.000, B 0.000, C 0.000 }
gfCNCPoint5[21479] = {X 415.7067, Y 102.1600, Z -7.1667, A 0.000, B 0.000, C 0.000 }
gfCNCPoint5[21480] = {X 396.4059, Y 102.1600, Z -7.1667, A 0.000, B 0.000, C 0.000 }
gfCNCPoint5[21481] = {X 395.4803, Y 102.0557, Z -7.1667, A 0.000, B 0.000, C 0.000 }
gfCNCPoint5[21482] = {X 394.6010, Y 101.7480, Z -7.1667, A 0.000, B 0.000, C 0.000 }
gfCNCPoint5[21483] = {X 393.8122, Y 101.2524, Z -7.1667, A 0.000, B 0.000, C 0.000 }
gfCNCPoint5[21484] = {X 393.1535, Y 100.5937, Z -7.1667, A 0.000, B 0.000, C 0.000 }
gfCNCPoint5[21485] = {X 392.6579, Y 99.8050, Z -7.1667, A 0.000, B 0.000, C 0.000 }
gfCNCPoint5[21486] = {X 392.3502, Y 98.9257, Z -7.1667, A 0.000, B 0.000, C 0.000 }
gfCNCPoint5[21487] = {X 392.2459, Y 98.0000, Z -7.1667, A 0.000, B 0.000, C 0.000 }
gfCNCPoint5[21488] = {X 392.2459, Y 97.0659, Z -7.1667, A 0.000, B 0.000, C 0.000 }
gfCNCPoint5[21489] = {X 392.3500, Y 96.1413, Z -7.1667, A 0.000, B 0.000, C 0.000 }
gfCNCPoint5[21490] = {X 392.6570, Y 95.2630, Z -7.1667, A 0.000, B 0.000, C 0.000 }
gfCNCPoint5[21491] = {X 393.1515, Y 94.4748, Z -7.1667, A 0.000, B 0.000, C 0.000 }
gfCNCPoint5[21492] = {X 393.8088, Y 93.8163, Z -7.1667, A 0.000, B 0.000, C 0.000 }
gfCNCPoint5[21493] = {X 394.5960, Y 93.3203, Z -7.1667, A 0.000, B 0.000, C 0.000 }
gfCNCPoint5[21494] = {X 395.4738, Y 93.0117, Z -7.1667, A 0.000, B 0.000, C 0.000 }
gfCNCPoint5[21495] = {X 396.3982, Y 92.9059, Z -7.1667, A 0.000, B 0.000, C 0.000 }
gfCNCPoint5[21496] = {X 397.3573, Y 92.8627, Z -7.1667, A 0.000, B 0.000, C 0.000 }
gfCNCPoint5[21497] = {X 398.3131, Y 92.7721, Z -7.1667, A 0.000, B 0.000, C 0.000 }
gfCNCPoint5[21498] = {X 398.9990, Y 92.6057, Z -7.1667, A 0.000, B 0.000, C 0.000 }
gfCNCPoint5[21499] = {X 399.6307, Y 92.2909, Z -7.1667, A 0.000, B 0.000, C 0.000 }
gfCNCPoint5[21500] = {X 413.8849, Y 83.1628, Z -7.1667, A 0.000, B 0.000, C 0.000 }
gfCNCPoint5[21501] = {X 411.7278, Y 79.7943, Z -7.1667, A 0.000, B 0.000, C 0.000 }
gfCNCPoint5[21502] = {X 413.9281, Y 83.2302, Z -7.1667, A 0.000, B 0.000, C 0.000 }
gfCNCPoint5[21503] = {X 428.5791, Y 73.8480, Z -7.1667, A 0.000, B 0.000, C 0.000 }
gfCNCPoint5[21504] = {X 403.8433, Y 64.1435, Z -7.1667, A 0.000, B 0.000, C 0.000 }
gfCNCPoint5[21505] = {X 402.1208, Y 63.5734, Z -7.1667, A 0.000, B 0.000, C 0.000 }
gfCNCPoint5[21506] = {X 400.3461, Y 63.1954, Z -7.1667, A 0.000, B 0.000, C 0.000 }
gfCNCPoint5[21507] = {X 398.5408, Y 63.0140, Z -7.1667, A 0.000, B 0.000, C 0.000 }
gfCNCPoint5[21508] = {X 397.6403, Y 62.9096, Z -7.1667, A 0.000, B 0.000, C 0.000 }
gfCNCPoint5[21509] = {X 396.7852, Y 62.6089, Z -7.1667, A 0.000, B 0.000, C 0.000 }
gfCNCPoint5[21510] = {X 396.0176, Y 62.1269, Z -7.1667, A 0.000, B 0.000, C 0.000 }
gfCNCPoint5[21511] = {X 395.3753, Y 61.4873, Z -7.1667, A 0.000, B 0.000, C 0.000 }
gfCNCPoint5[21512] = {X 394.8901, Y 60.7216, Z -7.1667, A 0.000, B 0.000, C 0.000 }
gfCNCPoint5[21513] = {X 394.5860, Y 59.8677, Z -7.1667, A 0.000, B 0.000, C 0.000 }
gfCNCPoint5[21514] = {X 394.4779, Y 58.9678, Z -7.1667, A 0.000, B 0.000, C 0.000 }
gfCNCPoint5[21515] = {X 394.4777, Y 58.0000, Z -7.1667, A 0.000, B 0.000, C 0.000 }
gfCNCPoint5[21516] = {X 394.5800, Y 57.0921, Z -7.1667, A 0.000, B 0.000, C 0.000 }
gfCNCPoint5[21517] = {X 394.8818, Y 56.2298, Z -7.1667, A 0.000, B 0.000, C 0.000 }
gfCNCPoint5[21518] = {X 395.3679, Y 55.4562, Z -7.1667, A 0.000, B 0.000, C 0.000 }
gfCNCPoint5[21519] = {X 396.0139, Y 54.8101, Z -7.1667, A 0.000, B 0.000, C 0.000 }
gfCNCPoint5[21520] = {X 396.7875, Y 54.3240, Z -7.1667, A 0.000, B 0.000, C 0.000 }
gfCNCPoint5[21521] = {X 397.6498, Y 54.0223, Z -7.1667, A 0.000, B 0.000, C 0.000 }
gfCNCPoint5[21522] = {X 398.5577, Y 53.9200, Z -7.1667, A 0.000, B 0.000, C 0.000 }
gfCNCPoint5[21523] = {X 419.4886, Y 53.9200, Z -7.1667, A 0.000, B 0.000, C 0.000 }
gfCNCPoint5[21524] = {X 420.3965, Y 54.0223, Z -7.1667, A 0.000, B 0.000, C 0.000 }
gfCNCPoint5[21525] = {X 421.2589, Y 54.3240, Z -7.1667, A 0.000, B 0.000, C 0.000 }
gfCNCPoint5[21526] = {X 422.0324, Y 54.8101, Z -7.1667, A 0.000, B 0.000, C 0.000 }
gfCNCPoint5[21527] = {X 422.6785, Y 55.4562, Z -7.1667, A 0.000, B 0.000, C 0.000 }
gfCNCPoint5[21528] = {X 423.1646, Y 56.2298, Z -7.1667, A 0.000, B 0.000, C 0.000 }
gfCNCPoint5[21529] = {X 423.4663, Y 57.0921, Z -7.1667, A 0.000, B 0.000, C 0.000 }
gfCNCPoint5[21530] = {X 423.5686, Y 58.0000, Z -7.1667, A 0.000, B 0.000, C 0.000 }
gfCNCPoint5[21531] = {X 423.5686, Y 58.3956, Z -7.1667, A 0.000, B 0.000, C 0.000 }
gfCNCPoint5[21532] = {X 429.5238, Y 60.7157, Z -7.1667, A 0.000, B 0.000, C 0.000 }
gfCNCPoint5[21533] = {X 458.0980, Y 72.0532, Z -7.1667, A 0.000, B 0.000, C 0.000 }
gfCNCPoint5[21534] = {X 458.1003, Y 62.9982, Z -7.1667, A 0.000, B 0.000, C 0.000 }
gfCNCPoint5[21535] = {X 457.9638, Y 62.9838, Z -7.1667, A 0.000, B 0.000, C 0.000 }
gfCNCPoint5[21536] = {X 457.8279, Y 62.9649, Z -7.1667, A 0.000, B 0.000, C 0.000 }
gfCNCPoint5[21537] = {X 456.9085, Y 62.7077, Z -7.1667, A 0.000, B 0.000, C 0.000 }
gfCNCPoint5[21538] = {X 456.0741, Y 62.2440, Z -7.1667, A 0.000, B 0.000, C 0.000 }
gfCNCPoint5[21539] = {X 455.3703, Y 61.5991, Z -7.1667, A 0.000, B 0.000, C 0.000 }
gfCNCPoint5[21540] = {X 454.8356, Y 60.8083, Z -7.1667, A 0.000, B 0.000, C 0.000 }
gfCNCPoint5[21541] = {X 454.4992, Y 59.9149, Z -7.1667, A 0.000, B 0.000, C 0.000 }
gfCNCPoint5[21542] = {X 454.3797, Y 58.9678, Z -7.1667, A 0.000, B 0.000, C 0.000 }
gfCNCPoint5[21543] = {X 454.3796, Y 58.0000, Z -7.1667, A 0.000, B 0.000, C 0.000 }
gfCNCPoint5[21544] = {X 454.4819, Y 57.0921, Z -7.1667, A 0.000, B 0.000, C 0.000 }
gfCNCPoint5[21545] = {X 454.7837, Y 56.2298, Z -7.1667, A 0.000, B 0.000, C 0.000 }
gfCNCPoint5[21546] = {X 455.2697, Y 55.4562, Z -7.1667, A 0.000, B 0.000, C 0.000 }
gfCNCPoint5[21547] = {X 455.9158, Y 54.8101, Z -7.1667, A 0.000, B 0.000, C 0.000 }
gfCNCPoint5[21548] = {X 456.6894, Y 54.3240, Z -7.1667, A 0.000, B 0.000, C 0.000 }
gfCNCPoint5[21549] = {X 457.5517, Y 54.0223, Z -7.1667, A 0.000, B 0.000, C 0.000 }
gfCNCPoint5[21550] = {X 458.4596, Y 53.9200, Z -7.1667, A 0.000, B 0.000, C 0.000 }
gfCNCPoint5[21551] = {X 475.0000, Y 53.9200, Z -7.1667, A 0.000, B 0.000, C 0.000 }
gfCNCPoint5[21552] = {X 475.9079, Y 54.0223, Z -7.1667, A 0.000, B 0.000, C 0.000 }
gfCNCPoint5[21553] = {X 476.7702, Y 54.3240, Z -7.1667, A 0.000, B 0.000, C 0.000 }
gfCNCPoint5[21554] = {X 477.5438, Y 54.8101, Z -7.1667, A 0.000, B 0.000, C 0.000 }
gfCNCPoint5[21555] = {X 478.1899, Y 55.4562, Z -7.1667, A 0.000, B 0.000, C 0.000 }
gfCNCPoint5[21556] = {X 478.6760, Y 56.2298, Z -7.1667, A 0.000, B 0.000, C 0.000 }
gfCNCPoint5[21557] = {X 478.9777, Y 57.0921, Z -7.1667, A 0.000, B 0.000, C 0.000 }
gfCNCPoint5[21558] = {X 479.0800, Y 58.0000, Z -7.1667, A 0.000, B 0.000, C 0.000 }
gfCNCPoint5[21559] = {X 479.0800, Y 58.9342, Z -7.1667, A 0.000, B 0.000, C 0.000 }
gfCNCPoint5[21560] = {X 478.9670, Y 59.8878, Z -7.1667, A 0.000, B 0.000, C 0.000 }
gfCNCPoint5[21561] = {X 478.6342, Y 60.7885, Z -7.1667, A 0.000, B 0.000, C 0.000 }
gfCNCPoint5[21562] = {X 478.1002, Y 61.5865, Z -7.1667, A 0.000, B 0.000, C 0.000 }
gfCNCPoint5[21563] = {X 477.3944, Y 62.2376, Z -7.1667, A 0.000, B 0.000, C 0.000 }
gfCNCPoint5[21564] = {X 476.5560, Y 62.7057, Z -7.1667, A 0.000, B 0.000, C 0.000 }
gfCNCPoint5[21565] = {X 475.6315, Y 62.9649, Z -7.1667, A 0.000, B 0.000, C 0.000 }
gfCNCPoint5[21566] = {X 475.4965, Y 62.9837, Z -7.1667, A 0.000, B 0.000, C 0.000 }
gfCNCPoint5[21567] = {X 475.3610, Y 62.9981, Z -7.1667, A 0.000, B 0.000, C 0.000 }
gfCNCPoint5[21568] = {X 475.3614, Y 92.9624, Z -7.1667, A 0.000, B 0.000, C 0.000 }
gfCNCPoint5[21569] = {X 475.8368, Y 93.0715, Z -7.1667, A 0.000, B 0.000, C 0.000 }
gfCNCPoint5[21570] = {X 476.3042, Y 93.2107, Z -7.1667, A 0.000, B 0.000, C 0.000 }
gfCNCPoint5[21571] = {X 477.0724, Y 93.5590, Z -7.1667, A 0.000, B 0.000, C 0.000 }
gfCNCPoint5[21572] = {X 477.7520, Y 94.0586, Z -7.1667, A 0.000, B 0.000, C 0.000 }
gfCNCPoint5[21573] = {X 478.3137, Y 94.6878, Z -7.1667, A 0.000, B 0.000, C 0.000 }
gfCNCPoint5[21574] = {X 478.7332, Y 95.4196, Z -7.1667, A 0.000, B 0.000, C 0.000 }
gfCNCPoint5[21575] = {X 478.9923, Y 96.2222, Z -7.1667, A 0.000, B 0.000, C 0.000 }
gfCNCPoint5[21576] = {X 479.0800, Y 97.0611, Z -7.1667, A 0.000, B 0.000, C 0.000 }
gfCNCPoint5[21577] = {X 479.0800, Y 98.0000, Z -7.1667, A 0.000, B 0.000, C 0.000 }
gfCNCPoint5[21578] = {X 478.9777, Y 98.9079, Z -7.1667, A 0.000, B 0.000, C 0.000 }
gfCNCPoint5[21579] = {X 478.6760, Y 99.7702, Z -7.1667, A 0.000, B 0.000, C 0.000 }
gfCNCPoint5[21580] = {X 478.1899, Y 100.5438, Z -7.1667, A 0.000, B 0.000, C 0.000 }
gfCNCPoint5[21581] = {X 477.5438, Y 101.1899, Z -7.1667, A 0.000, B 0.000, C 0.000 }
gfCNCPoint5[21582] = {X 476.7702, Y 101.6760, Z -7.1667, A 0.000, B 0.000, C 0.000 }
gfCNCPoint5[21583] = {X 475.9079, Y 101.9777, Z -7.1667, A 0.000, B 0.000, C 0.000 }
gfCNCPoint5[21584] = {X 475.0000, Y 102.0800, Z -7.1667, A 0.000, B 0.000, C 0.000 }
gfCNCPoint5[21585] = {X 458.4596, Y 102.0800, Z -7.1667, A 0.000, B 0.000, C 0.000 }
gfCNCPoint5[21586] = {X 457.5517, Y 101.9777, Z -7.1667, A 0.000, B 0.000, C 0.000 }
gfCNCPoint5[21587] = {X 456.6894, Y 101.6760, Z -7.1667, A 0.000, B 0.000, C 0.000 }
gfCNCPoint5[21588] = {X 455.9158, Y 101.1899, Z -7.1667, A 0.000, B 0.000, C 0.000 }
gfCNCPoint5[21589] = {X 455.2697, Y 100.5438, Z -7.1667, A 0.000, B 0.000, C 0.000 }
gfCNCPoint5[21590] = {X 454.7837, Y 99.7702, Z -7.1667, A 0.000, B 0.000, C 0.000 }
gfCNCPoint5[21591] = {X 454.4819, Y 98.9079, Z -7.1667, A 0.000, B 0.000, C 0.000 }
gfCNCPoint5[21592] = {X 454.3796, Y 98.0000, Z -7.1667, A 0.000, B 0.000, C 0.000 }
gfCNCPoint5[21593] = {X 454.3796, Y 97.0659, Z -7.1667, A 0.000, B 0.000, C 0.000 }
gfCNCPoint5[21594] = {X 454.4707, Y 96.2088, Z -7.1667, A 0.000, B 0.000, C 0.000 }
gfCNCPoint5[21595] = {X 454.7398, Y 95.3899, Z -7.1667, A 0.000, B 0.000, C 0.000 }
gfCNCPoint5[21596] = {X 455.1749, Y 94.6458, Z -7.1667, A 0.000, B 0.000, C 0.000 }
gfCNCPoint5[21597] = {X 455.7566, Y 94.0098, Z -7.1667, A 0.000, B 0.000, C 0.000 }
gfCNCPoint5[21598] = {X 456.4590, Y 93.5101, Z -7.1667, A 0.000, B 0.000, C 0.000 }
gfCNCPoint5[21599] = {X 457.2507, Y 93.1692, Z -7.1667, A 0.000, B 0.000, C 0.000 }
gfCNCPoint5[21600] = {X 458.0963, Y 93.0021, Z -7.1667, A 0.000, B 0.000, C 0.000 }
gfCNCPoint5[21601] = {X 458.0963, Y 85.4313, Z -7.1667, A 0.000, B 0.000, C 0.000 }
gfCNCPoint5[21602] = {X 444.8331, Y 80.2321, Z -7.1667, A 0.000, B 0.000, C 0.000 }
gfCNCPoint5[21603] = {X 419.7835, Y 96.4584, Z -7.1667, A 0.000, B 0.000, C 0.000 }
gfCNCPoint5[21604] = {X 419.7867, Y 97.0657, Z -7.1667, A 0.000, B 0.000, C 0.000 }
gfCNCPoint5[21605] = {X 419.7867, Y 98.0000, Z -7.1667, A 0.000, B 0.000, C 0.000 }
gfCNCPoint5[21606] = {X 419.6844, Y 98.9079, Z -7.1667, A 0.000, B 0.000, C 0.000 }
gfCNCPoint5[21607] = {X 419.3827, Y 99.7702, Z -7.1667, A 0.000, B 0.000, C 0.000 }
gfCNCPoint5[21608] = {X 418.8966, Y 100.5438, Z -7.1667, A 0.000, B 0.000, C 0.000 }
gfCNCPoint5[21609] = {X 418.2505, Y 101.1899, Z -7.1667, A 0.000, B 0.000, C 0.000 }
gfCNCPoint5[21610] = {X 417.4769, Y 101.6760, Z -7.1667, A 0.000, B 0.000, C 0.000 }
